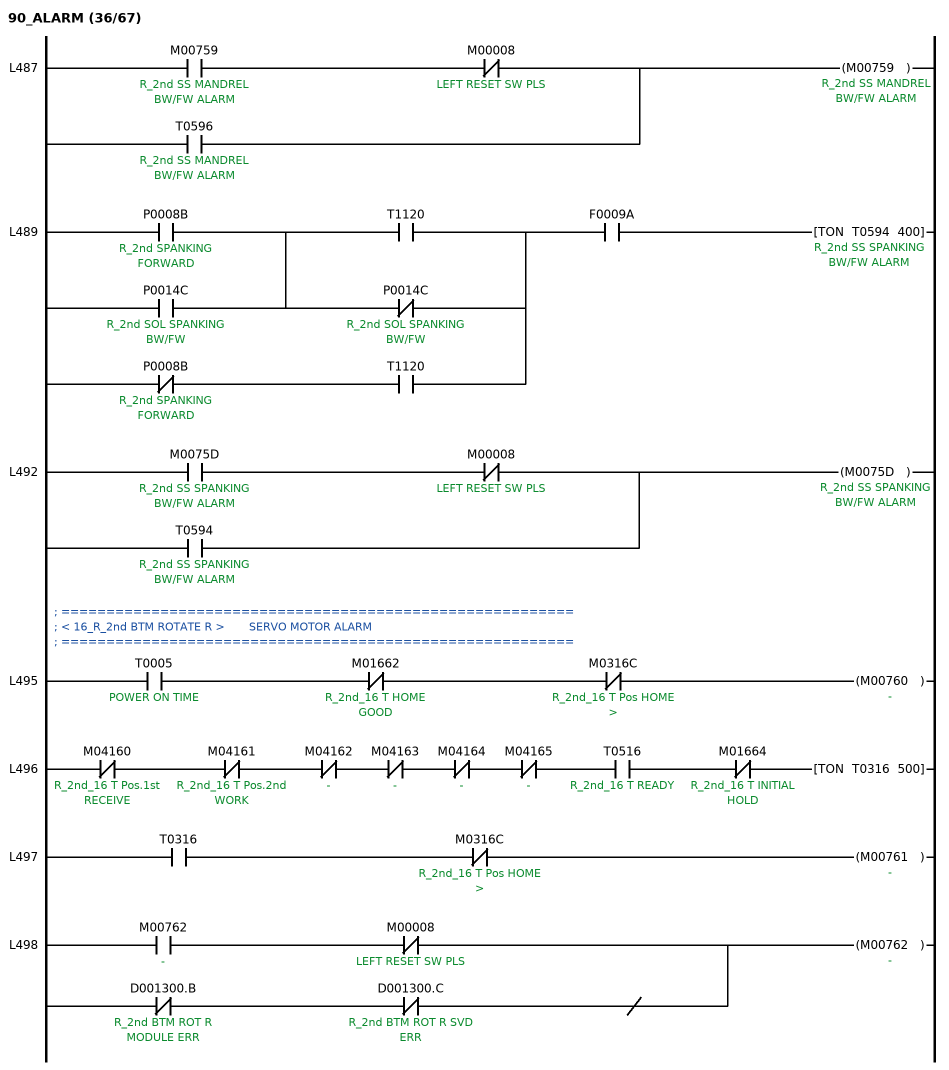
[picture p432: 90_ALARM rungs L487-L498]
; L487
LOAD      M00759	// R_2nd SS MANDREL BW/FW ALARM
AND NOT   M00008	// LEFT RESET SW PLS
OR        T0596	// R_2nd SS MANDREL BW/FW ALARM
OUT       M00759	// R_2nd SS MANDREL BW/FW ALARM
; L489
LOAD      P0008B	// R_2nd SPANKING FORWARD
OR        P0014C	// R_2nd SOL SPANKING BW/FW
LOAD      T1120
OR NOT    P0014C	// R_2nd SOL SPANKING BW/FW
AND LOAD
LOAD NOT  P0008B	// R_2nd SPANKING FORWARD
AND       T1120
OR LOAD
AND       F0009A
TON       T0594 400	// R_2nd SS SPANKING BW/FW ALARM
; L492
LOAD      M0075D	// R_2nd SS SPANKING BW/FW ALARM
AND NOT   M00008	// LEFT RESET SW PLS
OR        T0594	// R_2nd SS SPANKING BW/FW ALARM
OUT       M0075D	// R_2nd SS SPANKING BW/FW ALARM
// =========================================================
// 
//        < 16_R_2nd BTM ROTATE R >       SERVO MOTOR ALARM
// 
// =========================================================
; L495
LOAD      T0005	// POWER ON TIME
AND NOT   M01662	// R_2nd_16 T HOME GOOD
AND NOT   M0316C	// R_2nd_16 T Pos HOME >
OUT       M00760	// -
; L496
LOAD NOT  M04160	// R_2nd_16 T Pos.1st RECEIVE
AND NOT   M04161	// R_2nd_16 T Pos.2nd WORK
AND NOT   M04162	// -
AND NOT   M04163	// -
AND NOT   M04164	// -
AND NOT   M04165	// -
AND       T0516	// R_2nd_16 T READY
AND NOT   M01664	// R_2nd_16 T INITIAL HOLD
TON       T0316 500
; L497
LOAD      T0316
AND NOT   M0316C	// R_2nd_16 T Pos HOME >
OUT       M00761	// -
; L498
LOAD      M00762	// -
AND NOT   M00008	// LEFT RESET SW PLS
LOAD NOT  D001300.B	// R_2nd BTM ROT R MODULE ERR
AND NOT   D001300.C	// R_2nd BTM ROT R SVD ERR
NOT
OR LOAD
OUT       M00762	// -

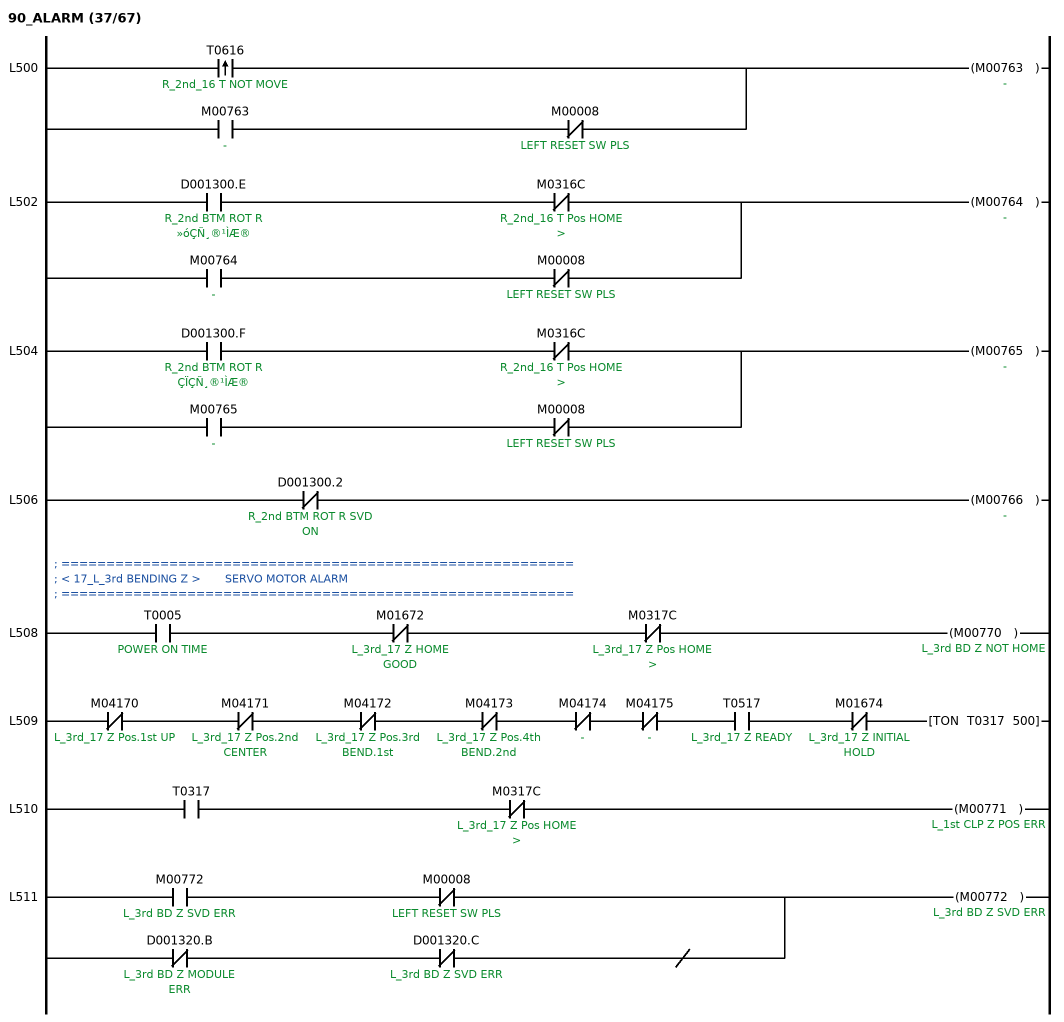
; L500
LOADP     T0616	// R_2nd_16 T NOT MOVE
LOAD      M00763	// -
AND NOT   M00008	// LEFT RESET SW PLS
OR LOAD
OUT       M00763	// -
; L502
LOAD      D001300.E	// R_2nd BTM ROT R »óÇÑ¸®¹ÌÆ®
AND NOT   M0316C	// R_2nd_16 T Pos HOME >
LOAD      M00764	// -
AND NOT   M00008	// LEFT RESET SW PLS
OR LOAD
OUT       M00764	// -
; L504
LOAD      D001300.F	// R_2nd BTM ROT R ÇÏÇÑ¸®¹ÌÆ®
AND NOT   M0316C	// R_2nd_16 T Pos HOME >
LOAD      M00765	// -
AND NOT   M00008	// LEFT RESET SW PLS
OR LOAD
OUT       M00765	// -
; L506
LOAD NOT  D001300.2	// R_2nd BTM ROT R SVD ON
OUT       M00766	// -
// =========================================================
// 
//        < 17_L_3rd BENDING Z >       SERVO MOTOR ALARM
// 
// =========================================================
; L508
LOAD      T0005	// POWER ON TIME
AND NOT   M01672	// L_3rd_17 Z HOME GOOD
AND NOT   M0317C	// L_3rd_17 Z Pos HOME >
OUT       M00770	// L_3rd BD Z NOT HOME
; L509
LOAD NOT  M04170	// L_3rd_17 Z Pos.1st UP
AND NOT   M04171	// L_3rd_17 Z Pos.2nd CENTER
AND NOT   M04172	// L_3rd_17 Z Pos.3rd BEND.1st
AND NOT   M04173	// L_3rd_17 Z Pos.4th BEND.2nd
AND NOT   M04174	// -
AND NOT   M04175	// -
AND       T0517	// L_3rd_17 Z READY
AND NOT   M01674	// L_3rd_17 Z INITIAL HOLD
TON       T0317 500
; L510
LOAD      T0317
AND NOT   M0317C	// L_3rd_17 Z Pos HOME >
OUT       M00771	// L_1st CLP Z POS ERR
; L511
LOAD      M00772	// L_3rd BD Z SVD ERR
AND NOT   M00008	// LEFT RESET SW PLS
LOAD NOT  D001320.B	// L_3rd BD Z MODULE ERR
AND NOT   D001320.C	// L_3rd BD Z SVD ERR
NOT
OR LOAD
OUT       M00772	// L_3rd BD Z SVD ERR

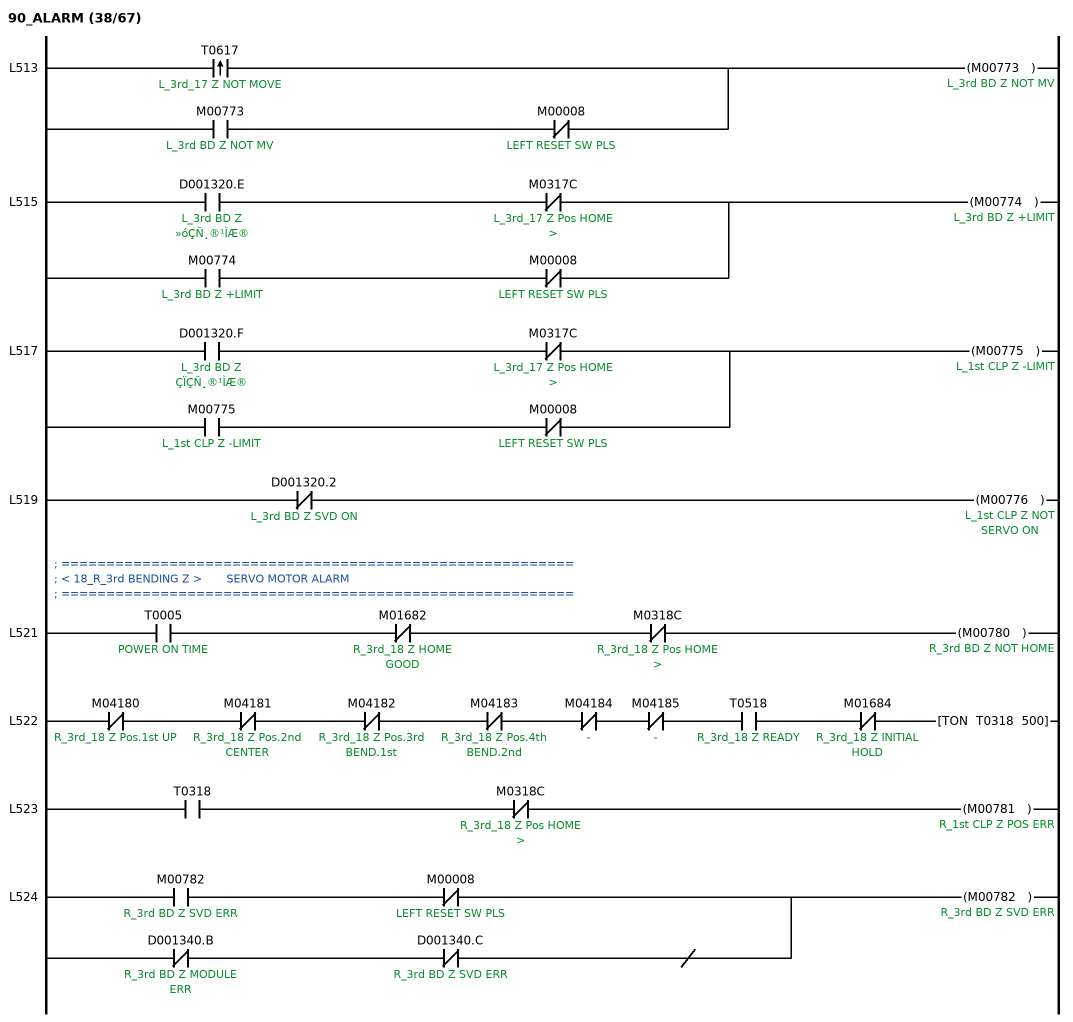
; L513
LOADP     T0617	// L_3rd_17 Z NOT MOVE
LOAD      M00773	// L_3rd BD Z NOT MV
AND NOT   M00008	// LEFT RESET SW PLS
OR LOAD
OUT       M00773	// L_3rd BD Z NOT MV
; L515
LOAD      D001320.E	// L_3rd BD Z »óÇÑ¸®¹ÌÆ®
AND NOT   M0317C	// L_3rd_17 Z Pos HOME >
LOAD      M00774	// L_3rd BD Z +LIMIT
AND NOT   M00008	// LEFT RESET SW PLS
OR LOAD
OUT       M00774	// L_3rd BD Z +LIMIT
; L517
LOAD      D001320.F	// L_3rd BD Z ÇÏÇÑ¸®¹ÌÆ®
AND NOT   M0317C	// L_3rd_17 Z Pos HOME >
LOAD      M00775	// L_1st CLP Z -LIMIT
AND NOT   M00008	// LEFT RESET SW PLS
OR LOAD
OUT       M00775	// L_1st CLP Z -LIMIT
; L519
LOAD NOT  D001320.2	// L_3rd BD Z SVD ON
OUT       M00776	// L_1st CLP Z NOT SERVO ON
// =========================================================
// 
//        < 18_R_3rd BENDING Z >       SERVO MOTOR ALARM
// 
// =========================================================
; L521
LOAD      T0005	// POWER ON TIME
AND NOT   M01682	// R_3rd_18 Z HOME GOOD
AND NOT   M0318C	// R_3rd_18 Z Pos HOME >
OUT       M00780	// R_3rd BD Z NOT HOME
; L522
LOAD NOT  M04180	// R_3rd_18 Z Pos.1st UP
AND NOT   M04181	// R_3rd_18 Z Pos.2nd CENTER
AND NOT   M04182	// R_3rd_18 Z Pos.3rd BEND.1st
AND NOT   M04183	// R_3rd_18 Z Pos.4th BEND.2nd
AND NOT   M04184	// -
AND NOT   M04185	// -
AND       T0518	// R_3rd_18 Z READY
AND NOT   M01684	// R_3rd_18 Z INITIAL HOLD
TON       T0318 500
; L523
LOAD      T0318
AND NOT   M0318C	// R_3rd_18 Z Pos HOME >
OUT       M00781	// R_1st CLP Z POS ERR
; L524
LOAD      M00782	// R_3rd BD Z SVD ERR
AND NOT   M00008	// LEFT RESET SW PLS
LOAD NOT  D001340.B	// R_3rd BD Z MODULE ERR
AND NOT   D001340.C	// R_3rd BD Z SVD ERR
NOT
OR LOAD
OUT       M00782	// R_3rd BD Z SVD ERR

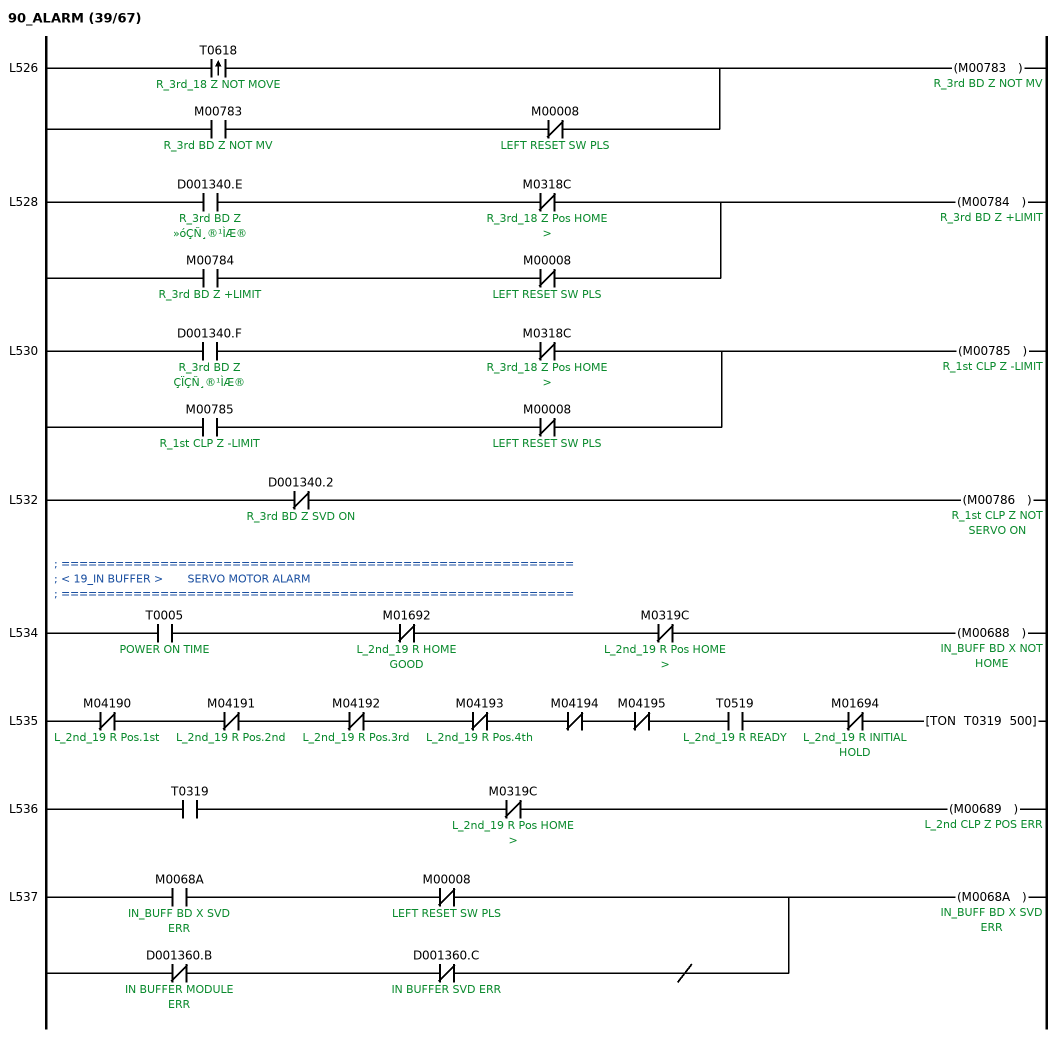
; L526
LOADP     T0618	// R_3rd_18 Z NOT MOVE
LOAD      M00783	// R_3rd BD Z NOT MV
AND NOT   M00008	// LEFT RESET SW PLS
OR LOAD
OUT       M00783	// R_3rd BD Z NOT MV
; L528
LOAD      D001340.E	// R_3rd BD Z »óÇÑ¸®¹ÌÆ®
AND NOT   M0318C	// R_3rd_18 Z Pos HOME >
LOAD      M00784	// R_3rd BD Z +LIMIT
AND NOT   M00008	// LEFT RESET SW PLS
OR LOAD
OUT       M00784	// R_3rd BD Z +LIMIT
; L530
LOAD      D001340.F	// R_3rd BD Z ÇÏÇÑ¸®¹ÌÆ®
AND NOT   M0318C	// R_3rd_18 Z Pos HOME >
LOAD      M00785	// R_1st CLP Z -LIMIT
AND NOT   M00008	// LEFT RESET SW PLS
OR LOAD
OUT       M00785	// R_1st CLP Z -LIMIT
; L532
LOAD NOT  D001340.2	// R_3rd BD Z SVD ON
OUT       M00786	// R_1st CLP Z NOT SERVO ON
// =========================================================
// 
//        < 19_IN BUFFER >       SERVO MOTOR ALARM
// 
// =========================================================
; L534
LOAD      T0005	// POWER ON TIME
AND NOT   M01692	// L_2nd_19 R HOME GOOD
AND NOT   M0319C	// L_2nd_19 R Pos HOME >
OUT       M00688	// IN_BUFF BD X NOT HOME
; L535
LOAD NOT  M04190	// L_2nd_19 R Pos.1st 
AND NOT   M04191	// L_2nd_19 R Pos.2nd
AND NOT   M04192	// L_2nd_19 R Pos.3rd
AND NOT   M04193	// L_2nd_19 R Pos.4th 
AND NOT   M04194
AND NOT   M04195
AND       T0519	// L_2nd_19 R READY
AND NOT   M01694	// L_2nd_19 R INITIAL HOLD
TON       T0319 500
; L536
LOAD      T0319
AND NOT   M0319C	// L_2nd_19 R Pos HOME >
OUT       M00689	// L_2nd CLP Z POS ERR
; L537
LOAD      M0068A	// IN_BUFF BD X SVD ERR
AND NOT   M00008	// LEFT RESET SW PLS
LOAD NOT  D001360.B	// IN BUFFER MODULE ERR
AND NOT   D001360.C	// IN BUFFER SVD ERR
NOT
OR LOAD
OUT       M0068A	// IN_BUFF BD X SVD ERR

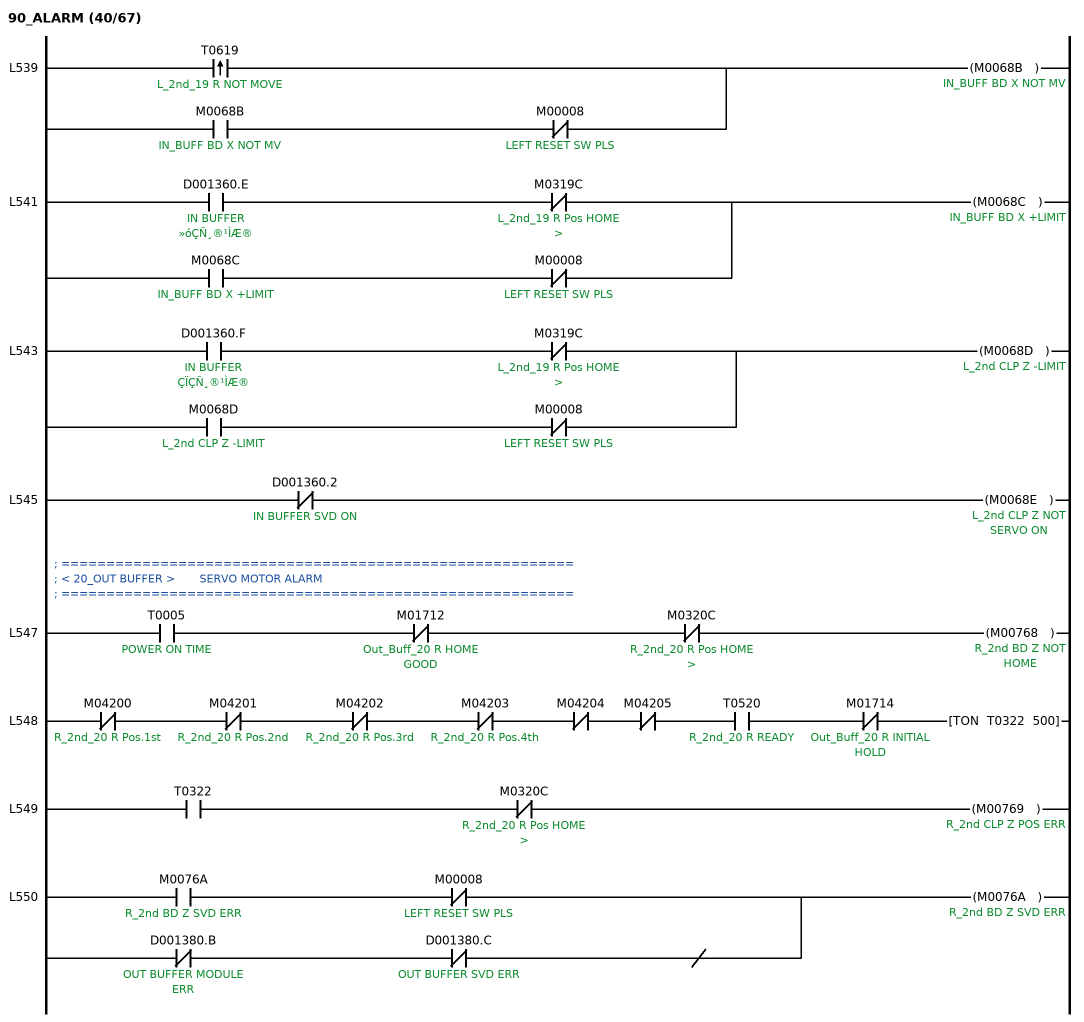
; L539
LOADP     T0619	// L_2nd_19 R NOT MOVE
LOAD      M0068B	// IN_BUFF BD X NOT MV
AND NOT   M00008	// LEFT RESET SW PLS
OR LOAD
OUT       M0068B	// IN_BUFF BD X NOT MV
; L541
LOAD      D001360.E	// IN BUFFER »óÇÑ¸®¹ÌÆ®
AND NOT   M0319C	// L_2nd_19 R Pos HOME >
LOAD      M0068C	// IN_BUFF BD X +LIMIT
AND NOT   M00008	// LEFT RESET SW PLS
OR LOAD
OUT       M0068C	// IN_BUFF BD X +LIMIT
; L543
LOAD      D001360.F	// IN BUFFER ÇÏÇÑ¸®¹ÌÆ®
AND NOT   M0319C	// L_2nd_19 R Pos HOME >
LOAD      M0068D	// L_2nd CLP Z -LIMIT
AND NOT   M00008	// LEFT RESET SW PLS
OR LOAD
OUT       M0068D	// L_2nd CLP Z -LIMIT
; L545
LOAD NOT  D001360.2	// IN BUFFER SVD ON
OUT       M0068E	// L_2nd CLP Z NOT SERVO ON
// =========================================================
// 
//        < 20_OUT BUFFER >       SERVO MOTOR ALARM
// 
// =========================================================
; L547
LOAD      T0005	// POWER ON TIME
AND NOT   M01712	// Out_Buff_20 R HOME GOOD
AND NOT   M0320C	// R_2nd_20 R Pos HOME >
OUT       M00768	// R_2nd BD Z NOT HOME
; L548
LOAD NOT  M04200	// R_2nd_20 R Pos.1st
AND NOT   M04201	// R_2nd_20 R Pos.2nd
AND NOT   M04202	// R_2nd_20 R Pos.3rd
AND NOT   M04203	// R_2nd_20 R Pos.4th 
AND NOT   M04204
AND NOT   M04205
AND       T0520	// R_2nd_20 R READY
AND NOT   M01714	// Out_Buff_20 R INITIAL HOLD
TON       T0322 500
; L549
LOAD      T0322
AND NOT   M0320C	// R_2nd_20 R Pos HOME >
OUT       M00769	// R_2nd CLP Z POS ERR
; L550
LOAD      M0076A	// R_2nd BD Z SVD ERR
AND NOT   M00008	// LEFT RESET SW PLS
LOAD NOT  D001380.B	// OUT BUFFER MODULE ERR
AND NOT   D001380.C	// OUT BUFFER SVD ERR
NOT
OR LOAD
OUT       M0076A	// R_2nd BD Z SVD ERR

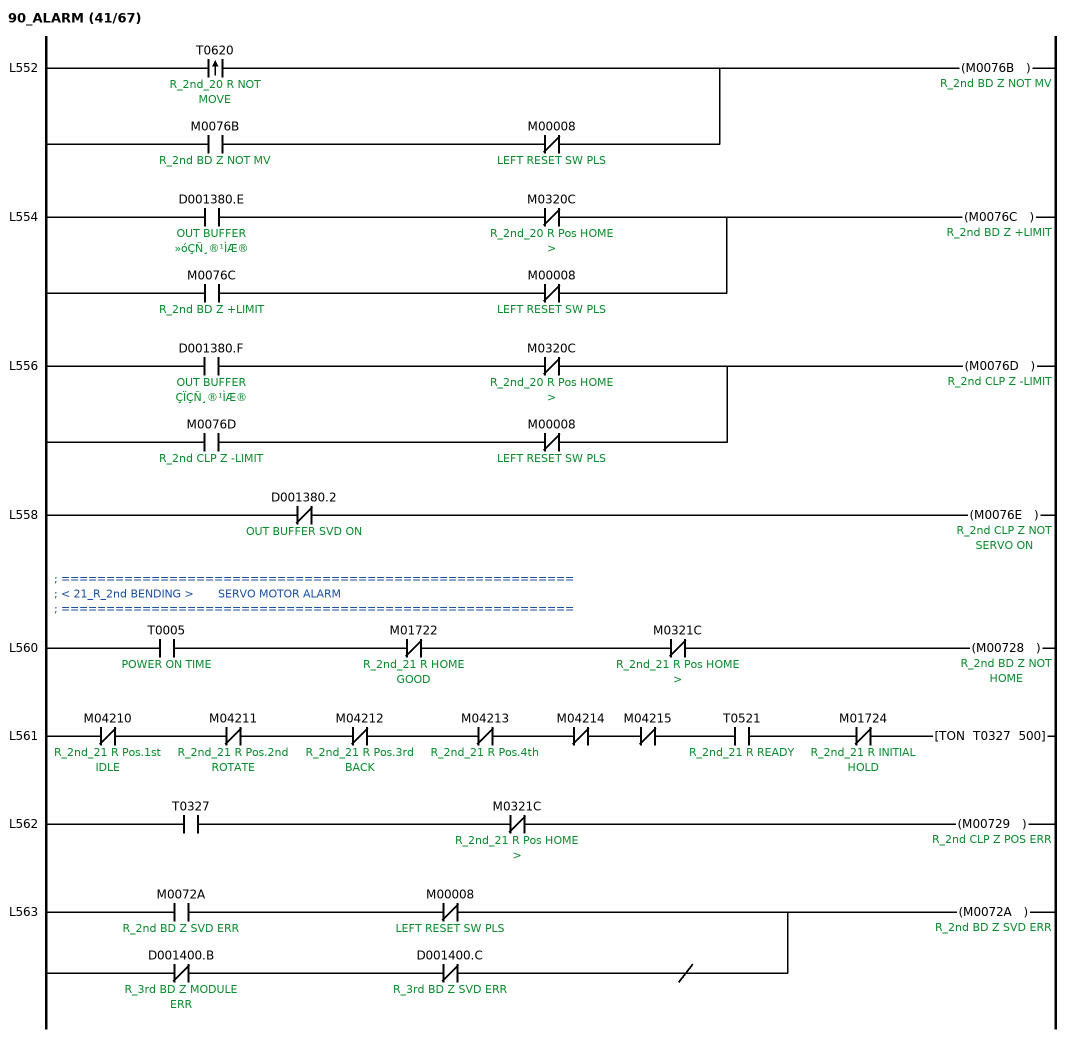
; L552
LOADP     T0620	// R_2nd_20 R NOT MOVE
LOAD      M0076B	// R_2nd BD Z NOT MV
AND NOT   M00008	// LEFT RESET SW PLS
OR LOAD
OUT       M0076B	// R_2nd BD Z NOT MV
; L554
LOAD      D001380.E	// OUT BUFFER »óÇÑ¸®¹ÌÆ®
AND NOT   M0320C	// R_2nd_20 R Pos HOME >
LOAD      M0076C	// R_2nd BD Z +LIMIT
AND NOT   M00008	// LEFT RESET SW PLS
OR LOAD
OUT       M0076C	// R_2nd BD Z +LIMIT
; L556
LOAD      D001380.F	// OUT BUFFER ÇÏÇÑ¸®¹ÌÆ®
AND NOT   M0320C	// R_2nd_20 R Pos HOME >
LOAD      M0076D	// R_2nd CLP Z -LIMIT
AND NOT   M00008	// LEFT RESET SW PLS
OR LOAD
OUT       M0076D	// R_2nd CLP Z -LIMIT
; L558
LOAD NOT  D001380.2	// OUT BUFFER SVD ON
OUT       M0076E	// R_2nd CLP Z NOT SERVO ON
// =========================================================
// 
//        < 21_R_2nd BENDING >       SERVO MOTOR ALARM
// 
// =========================================================
; L560
LOAD      T0005	// POWER ON TIME
AND NOT   M01722	// R_2nd_21 R HOME GOOD
AND NOT   M0321C	// R_2nd_21 R Pos HOME >
OUT       M00728	// R_2nd BD Z NOT HOME
; L561
LOAD NOT  M04210	// R_2nd_21 R Pos.1st IDLE
AND NOT   M04211	// R_2nd_21 R Pos.2nd ROTATE
AND NOT   M04212	// R_2nd_21 R Pos.3rd BACK
AND NOT   M04213	// R_2nd_21 R Pos.4th 
AND NOT   M04214
AND NOT   M04215
AND       T0521	// R_2nd_21 R READY
AND NOT   M01724	// R_2nd_21 R INITIAL HOLD
TON       T0327 500
; L562
LOAD      T0327
AND NOT   M0321C	// R_2nd_21 R Pos HOME >
OUT       M00729	// R_2nd CLP Z POS ERR
; L563
LOAD      M0072A	// R_2nd BD Z SVD ERR
AND NOT   M00008	// LEFT RESET SW PLS
LOAD NOT  D001400.B	// R_3rd BD Z MODULE ERR
AND NOT   D001400.C	// R_3rd BD Z SVD ERR
NOT
OR LOAD
OUT       M0072A	// R_2nd BD Z SVD ERR

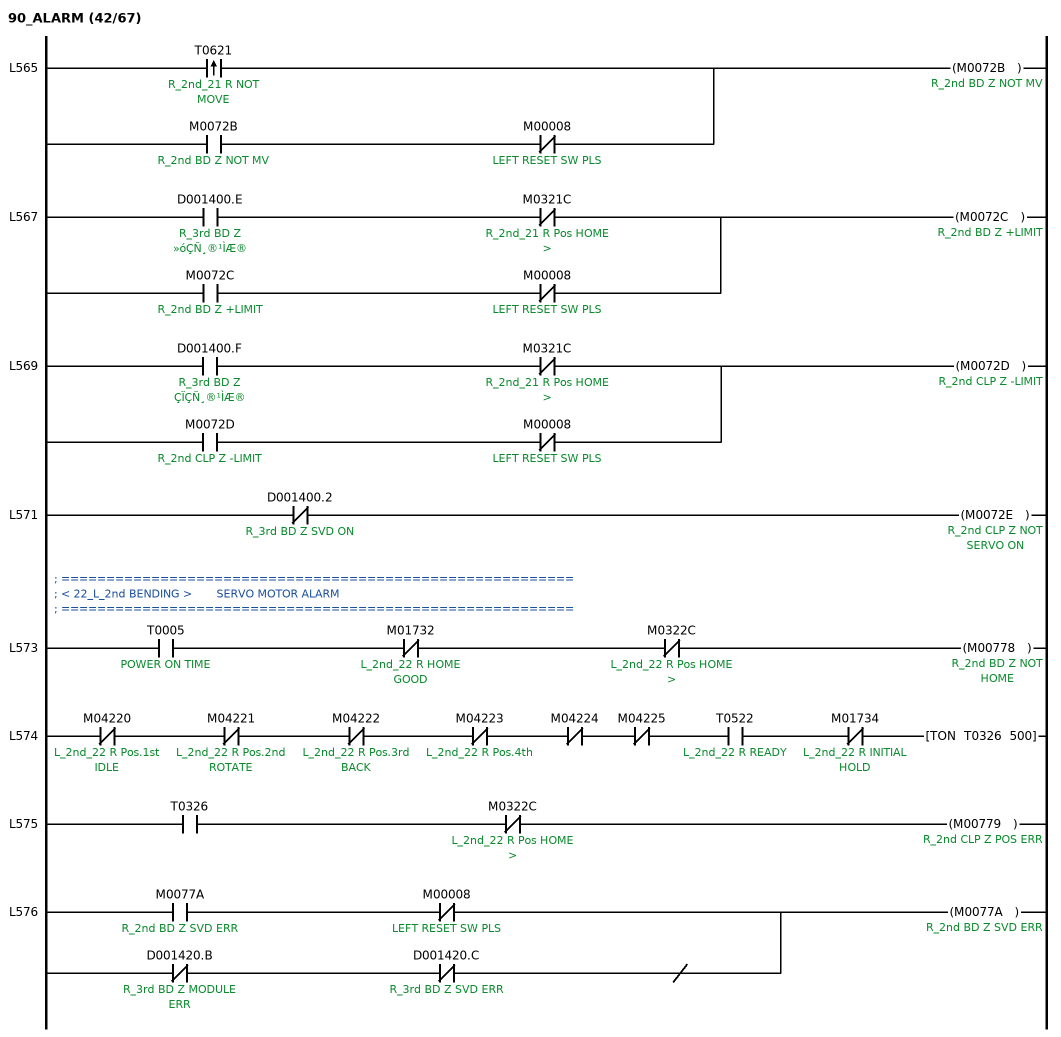
; L565
LOADP     T0621	// R_2nd_21 R NOT MOVE
LOAD      M0072B	// R_2nd BD Z NOT MV
AND NOT   M00008	// LEFT RESET SW PLS
OR LOAD
OUT       M0072B	// R_2nd BD Z NOT MV
; L567
LOAD      D001400.E	// R_3rd BD Z »óÇÑ¸®¹ÌÆ®
AND NOT   M0321C	// R_2nd_21 R Pos HOME >
LOAD      M0072C	// R_2nd BD Z +LIMIT
AND NOT   M00008	// LEFT RESET SW PLS
OR LOAD
OUT       M0072C	// R_2nd BD Z +LIMIT
; L569
LOAD      D001400.F	// R_3rd BD Z ÇÏÇÑ¸®¹ÌÆ®
AND NOT   M0321C	// R_2nd_21 R Pos HOME >
LOAD      M0072D	// R_2nd CLP Z -LIMIT
AND NOT   M00008	// LEFT RESET SW PLS
OR LOAD
OUT       M0072D	// R_2nd CLP Z -LIMIT
; L571
LOAD NOT  D001400.2	// R_3rd BD Z SVD ON
OUT       M0072E	// R_2nd CLP Z NOT SERVO ON
// =========================================================
// 
//        < 22_L_2nd BENDING >       SERVO MOTOR ALARM
// 
// =========================================================
; L573
LOAD      T0005	// POWER ON TIME
AND NOT   M01732	// L_2nd_22 R HOME GOOD
AND NOT   M0322C	// L_2nd_22 R Pos HOME >
OUT       M00778	// R_2nd BD Z NOT HOME
; L574
LOAD NOT  M04220	// L_2nd_22 R Pos.1st IDLE
AND NOT   M04221	// L_2nd_22 R Pos.2nd ROTATE
AND NOT   M04222	// L_2nd_22 R Pos.3rd BACK
AND NOT   M04223	// L_2nd_22 R Pos.4th 
AND NOT   M04224
AND NOT   M04225
AND       T0522	// L_2nd_22 R READY
AND NOT   M01734	// L_2nd_22 R INITIAL HOLD
TON       T0326 500
; L575
LOAD      T0326
AND NOT   M0322C	// L_2nd_22 R Pos HOME >
OUT       M00779	// R_2nd CLP Z POS ERR
; L576
LOAD      M0077A	// R_2nd BD Z SVD ERR
AND NOT   M00008	// LEFT RESET SW PLS
LOAD NOT  D001420.B	// R_3rd BD Z MODULE ERR
AND NOT   D001420.C	// R_3rd BD Z SVD ERR
NOT
OR LOAD
OUT       M0077A	// R_2nd BD Z SVD ERR

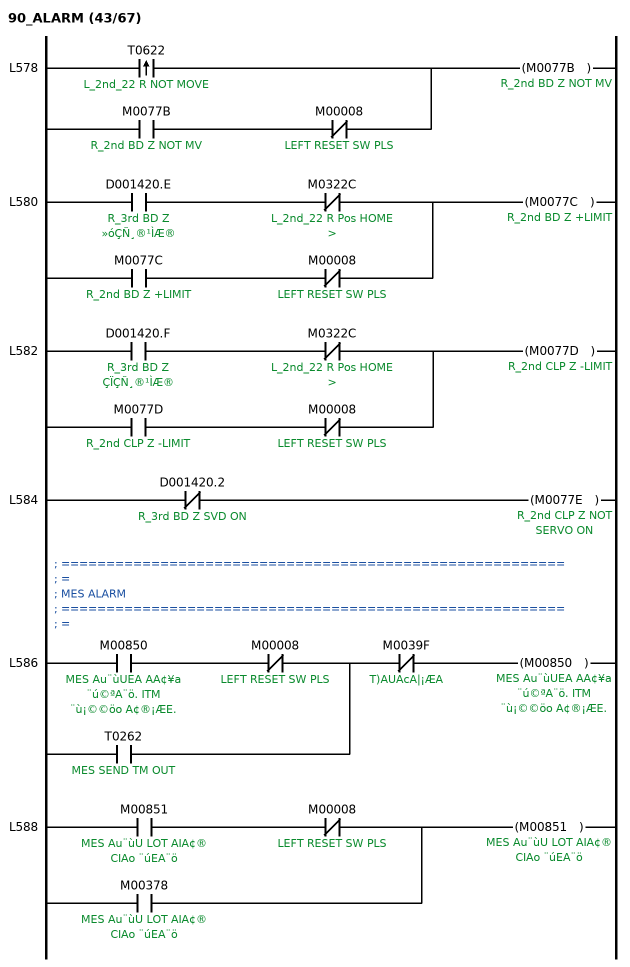
; L578
LOADP     T0622	// L_2nd_22 R NOT MOVE
LOAD      M0077B	// R_2nd BD Z NOT MV
AND NOT   M00008	// LEFT RESET SW PLS
OR LOAD
OUT       M0077B	// R_2nd BD Z NOT MV
; L580
LOAD      D001420.E	// R_3rd BD Z »óÇÑ¸®¹ÌÆ®
AND NOT   M0322C	// L_2nd_22 R Pos HOME >
LOAD      M0077C	// R_2nd BD Z +LIMIT
AND NOT   M00008	// LEFT RESET SW PLS
OR LOAD
OUT       M0077C	// R_2nd BD Z +LIMIT
; L582
LOAD      D001420.F	// R_3rd BD Z ÇÏÇÑ¸®¹ÌÆ®
AND NOT   M0322C	// L_2nd_22 R Pos HOME >
LOAD      M0077D	// R_2nd CLP Z -LIMIT
AND NOT   M00008	// LEFT RESET SW PLS
OR LOAD
OUT       M0077D	// R_2nd CLP Z -LIMIT
; L584
LOAD NOT  D001420.2	// R_3rd BD Z SVD ON
OUT       M0077E	// R_2nd CLP Z NOT SERVO ON
// =========================================================
// 
//        MES ALARM
// 
// =========================================================
; L586
LOAD      M00850	// MES Au¨ùUEA AA¢¥a ¨ú©ªA¨ö. ITM ¨ù¡©©öo A¢®¡ÆE.
AND NOT   M00008	// LEFT RESET SW PLS
OR        T0262	// MES SEND TM OUT
AND NOT   M0039F	// T)AUAcA|¡ÆA
OUT       M00850	// MES Au¨ùUEA AA¢¥a ¨ú©ªA¨ö. ITM ¨ù¡©©öo A¢®¡ÆE.
; L588
LOAD      M00851	// MES Au¨ùU LOT AIA¢® CIAo ¨úEA¨ö
AND NOT   M00008	// LEFT RESET SW PLS
OR        M00378	// MES Au¨ùU LOT AIA¢® CIAo ¨úEA¨ö
OUT       M00851	// MES Au¨ùU LOT AIA¢® CIAo ¨úEA¨ö

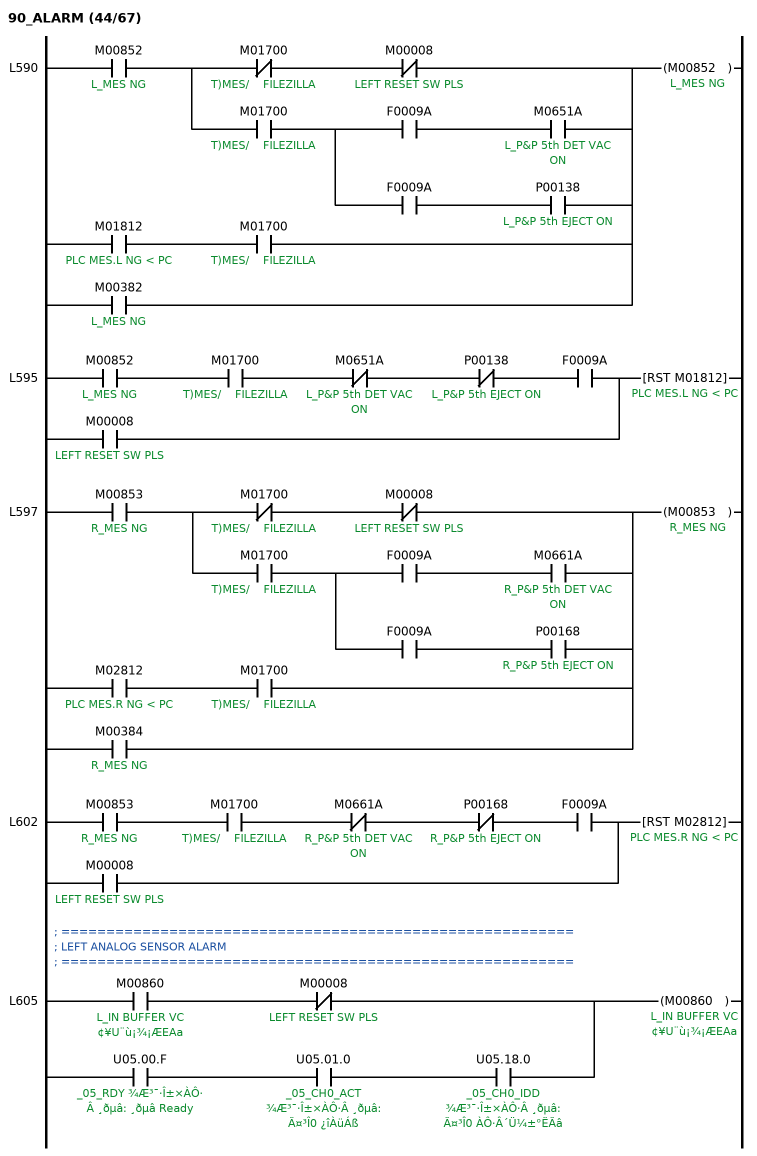
; L590
LOAD      M00852	// L_MES NG
LOAD NOT  M01700	// T)MES/    FILEZILLA
AND NOT   M00008	// LEFT RESET SW PLS
LOAD      M01700	// T)MES/    FILEZILLA
LOAD      F0009A
AND       M0651A	// L_P&P 5th DET VAC ON
LOAD      F0009A
AND       P00138	// L_P&P 5th EJECT ON
OR LOAD
AND LOAD
OR LOAD
AND LOAD
LOAD      M01812	// PLC MES.L NG < PC
AND       M01700	// T)MES/    FILEZILLA
OR LOAD
OR        M00382	// L_MES NG
OUT       M00852	// L_MES NG
; L595
LOAD      M00852	// L_MES NG
AND       M01700	// T)MES/    FILEZILLA
AND NOT   M0651A	// L_P&P 5th DET VAC ON
AND NOT   P00138	// L_P&P 5th EJECT ON
AND       F0009A
OR        M00008	// LEFT RESET SW PLS
RST       M01812	// PLC MES.L NG < PC
; L597
LOAD      M00853	// R_MES NG
LOAD NOT  M01700	// T)MES/    FILEZILLA
AND NOT   M00008	// LEFT RESET SW PLS
LOAD      M01700	// T)MES/    FILEZILLA
LOAD      F0009A
AND       M0661A	// R_P&P 5th DET VAC ON
LOAD      F0009A
AND       P00168	// R_P&P 5th EJECT ON
OR LOAD
AND LOAD
OR LOAD
AND LOAD
LOAD      M02812	// PLC MES.R NG < PC
AND       M01700	// T)MES/    FILEZILLA
OR LOAD
OR        M00384	// R_MES NG
OUT       M00853	// R_MES NG
; L602
LOAD      M00853	// R_MES NG
AND       M01700	// T)MES/    FILEZILLA
AND NOT   M0661A	// R_P&P 5th DET VAC ON
AND NOT   P00168	// R_P&P 5th EJECT ON
AND       F0009A
OR        M00008	// LEFT RESET SW PLS
RST       M02812	// PLC MES.R NG < PC
// =========================================================
// 
//        LEFT ANALOG SENSOR ALARM
// 
// =========================================================
; L605
LOAD      M00860	// L_IN BUFFER VC ¢¥U¨ù¡¾¡ÆEAa
AND NOT   M00008	// LEFT RESET SW PLS
LOAD      U05.00.F	// _05_RDY ¾Æ³¯·Î±×ÀÔ·Â ¸ðµâ: ¸ðµâ Ready
AND       U05.01.0	// _05_CH0_ACT ¾Æ³¯·Î±×ÀÔ·Â ¸ðµâ: Ã¤³Î0 ¿îÀüÁß
AND       U05.18.0	// _05_CH0_IDD ¾Æ³¯·Î±×ÀÔ·Â ¸ðµâ: Ã¤³Î0 ÀÔ·Â´Ü¼±°ËÃâ
OR LOAD
OUT       M00860	// L_IN BUFFER VC ¢¥U¨ù¡¾¡ÆEAa

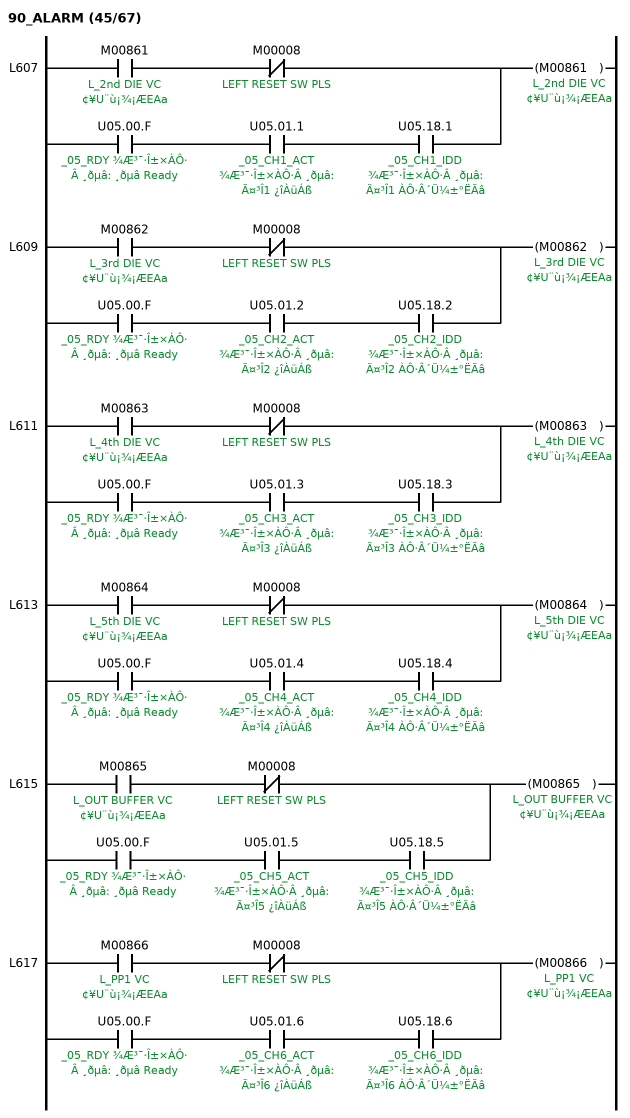
; L607
LOAD      M00861	// L_2nd DIE VC ¢¥U¨ù¡¾¡ÆEAa
AND NOT   M00008	// LEFT RESET SW PLS
LOAD      U05.00.F	// _05_RDY ¾Æ³¯·Î±×ÀÔ·Â ¸ðµâ: ¸ðµâ Ready
AND       U05.01.1	// _05_CH1_ACT ¾Æ³¯·Î±×ÀÔ·Â ¸ðµâ: Ã¤³Î1 ¿îÀüÁß
AND       U05.18.1	// _05_CH1_IDD ¾Æ³¯·Î±×ÀÔ·Â ¸ðµâ: Ã¤³Î1 ÀÔ·Â´Ü¼±°ËÃâ
OR LOAD
OUT       M00861	// L_2nd DIE VC ¢¥U¨ù¡¾¡ÆEAa
; L609
LOAD      M00862	// L_3rd DIE VC ¢¥U¨ù¡¾¡ÆEAa
AND NOT   M00008	// LEFT RESET SW PLS
LOAD      U05.00.F	// _05_RDY ¾Æ³¯·Î±×ÀÔ·Â ¸ðµâ: ¸ðµâ Ready
AND       U05.01.2	// _05_CH2_ACT ¾Æ³¯·Î±×ÀÔ·Â ¸ðµâ: Ã¤³Î2 ¿îÀüÁß
AND       U05.18.2	// _05_CH2_IDD ¾Æ³¯·Î±×ÀÔ·Â ¸ðµâ: Ã¤³Î2 ÀÔ·Â´Ü¼±°ËÃâ
OR LOAD
OUT       M00862	// L_3rd DIE VC ¢¥U¨ù¡¾¡ÆEAa
; L611
LOAD      M00863	// L_4th DIE VC ¢¥U¨ù¡¾¡ÆEAa
AND NOT   M00008	// LEFT RESET SW PLS
LOAD      U05.00.F	// _05_RDY ¾Æ³¯·Î±×ÀÔ·Â ¸ðµâ: ¸ðµâ Ready
AND       U05.01.3	// _05_CH3_ACT ¾Æ³¯·Î±×ÀÔ·Â ¸ðµâ: Ã¤³Î3 ¿îÀüÁß
AND       U05.18.3	// _05_CH3_IDD ¾Æ³¯·Î±×ÀÔ·Â ¸ðµâ: Ã¤³Î3 ÀÔ·Â´Ü¼±°ËÃâ
OR LOAD
OUT       M00863	// L_4th DIE VC ¢¥U¨ù¡¾¡ÆEAa
; L613
LOAD      M00864	// L_5th DIE VC ¢¥U¨ù¡¾¡ÆEAa
AND NOT   M00008	// LEFT RESET SW PLS
LOAD      U05.00.F	// _05_RDY ¾Æ³¯·Î±×ÀÔ·Â ¸ðµâ: ¸ðµâ Ready
AND       U05.01.4	// _05_CH4_ACT ¾Æ³¯·Î±×ÀÔ·Â ¸ðµâ: Ã¤³Î4 ¿îÀüÁß
AND       U05.18.4	// _05_CH4_IDD ¾Æ³¯·Î±×ÀÔ·Â ¸ðµâ: Ã¤³Î4 ÀÔ·Â´Ü¼±°ËÃâ
OR LOAD
OUT       M00864	// L_5th DIE VC ¢¥U¨ù¡¾¡ÆEAa
; L615
LOAD      M00865	// L_OUT BUFFER VC ¢¥U¨ù¡¾¡ÆEAa
AND NOT   M00008	// LEFT RESET SW PLS
LOAD      U05.00.F	// _05_RDY ¾Æ³¯·Î±×ÀÔ·Â ¸ðµâ: ¸ðµâ Ready
AND       U05.01.5	// _05_CH5_ACT ¾Æ³¯·Î±×ÀÔ·Â ¸ðµâ: Ã¤³Î5 ¿îÀüÁß
AND       U05.18.5	// _05_CH5_IDD ¾Æ³¯·Î±×ÀÔ·Â ¸ðµâ: Ã¤³Î5 ÀÔ·Â´Ü¼±°ËÃâ
OR LOAD
OUT       M00865	// L_OUT BUFFER VC ¢¥U¨ù¡¾¡ÆEAa
; L617
LOAD      M00866	// L_PP1 VC ¢¥U¨ù¡¾¡ÆEAa
AND NOT   M00008	// LEFT RESET SW PLS
LOAD      U05.00.F	// _05_RDY ¾Æ³¯·Î±×ÀÔ·Â ¸ðµâ: ¸ðµâ Ready
AND       U05.01.6	// _05_CH6_ACT ¾Æ³¯·Î±×ÀÔ·Â ¸ðµâ: Ã¤³Î6 ¿îÀüÁß
AND       U05.18.6	// _05_CH6_IDD ¾Æ³¯·Î±×ÀÔ·Â ¸ðµâ: Ã¤³Î6 ÀÔ·Â´Ü¼±°ËÃâ
OR LOAD
OUT       M00866	// L_PP1 VC ¢¥U¨ù¡¾¡ÆEAa

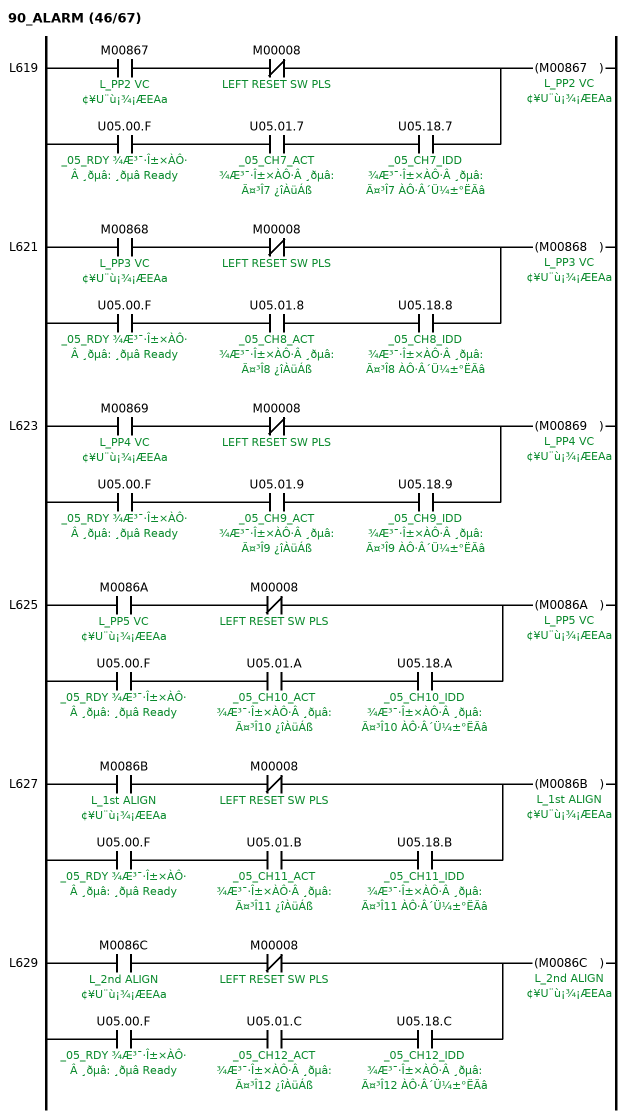
; L619
LOAD      M00867	// L_PP2 VC ¢¥U¨ù¡¾¡ÆEAa
AND NOT   M00008	// LEFT RESET SW PLS
LOAD      U05.00.F	// _05_RDY ¾Æ³¯·Î±×ÀÔ·Â ¸ðµâ: ¸ðµâ Ready
AND       U05.01.7	// _05_CH7_ACT ¾Æ³¯·Î±×ÀÔ·Â ¸ðµâ: Ã¤³Î7 ¿îÀüÁß
AND       U05.18.7	// _05_CH7_IDD ¾Æ³¯·Î±×ÀÔ·Â ¸ðµâ: Ã¤³Î7 ÀÔ·Â´Ü¼±°ËÃâ
OR LOAD
OUT       M00867	// L_PP2 VC ¢¥U¨ù¡¾¡ÆEAa
; L621
LOAD      M00868	// L_PP3 VC ¢¥U¨ù¡¾¡ÆEAa
AND NOT   M00008	// LEFT RESET SW PLS
LOAD      U05.00.F	// _05_RDY ¾Æ³¯·Î±×ÀÔ·Â ¸ðµâ: ¸ðµâ Ready
AND       U05.01.8	// _05_CH8_ACT ¾Æ³¯·Î±×ÀÔ·Â ¸ðµâ: Ã¤³Î8 ¿îÀüÁß
AND       U05.18.8	// _05_CH8_IDD ¾Æ³¯·Î±×ÀÔ·Â ¸ðµâ: Ã¤³Î8 ÀÔ·Â´Ü¼±°ËÃâ
OR LOAD
OUT       M00868	// L_PP3 VC ¢¥U¨ù¡¾¡ÆEAa
; L623
LOAD      M00869	// L_PP4 VC ¢¥U¨ù¡¾¡ÆEAa
AND NOT   M00008	// LEFT RESET SW PLS
LOAD      U05.00.F	// _05_RDY ¾Æ³¯·Î±×ÀÔ·Â ¸ðµâ: ¸ðµâ Ready
AND       U05.01.9	// _05_CH9_ACT ¾Æ³¯·Î±×ÀÔ·Â ¸ðµâ: Ã¤³Î9 ¿îÀüÁß
AND       U05.18.9	// _05_CH9_IDD ¾Æ³¯·Î±×ÀÔ·Â ¸ðµâ: Ã¤³Î9 ÀÔ·Â´Ü¼±°ËÃâ
OR LOAD
OUT       M00869	// L_PP4 VC ¢¥U¨ù¡¾¡ÆEAa
; L625
LOAD      M0086A	// L_PP5 VC ¢¥U¨ù¡¾¡ÆEAa
AND NOT   M00008	// LEFT RESET SW PLS
LOAD      U05.00.F	// _05_RDY ¾Æ³¯·Î±×ÀÔ·Â ¸ðµâ: ¸ðµâ Ready
AND       U05.01.A	// _05_CH10_ACT ¾Æ³¯·Î±×ÀÔ·Â ¸ðµâ: Ã¤³Î10 ¿îÀüÁß
AND       U05.18.A	// _05_CH10_IDD ¾Æ³¯·Î±×ÀÔ·Â ¸ðµâ: Ã¤³Î10 ÀÔ·Â´Ü¼±°ËÃâ
OR LOAD
OUT       M0086A	// L_PP5 VC ¢¥U¨ù¡¾¡ÆEAa
; L627
LOAD      M0086B	// L_1st ALIGN ¢¥U¨ù¡¾¡ÆEAa
AND NOT   M00008	// LEFT RESET SW PLS
LOAD      U05.00.F	// _05_RDY ¾Æ³¯·Î±×ÀÔ·Â ¸ðµâ: ¸ðµâ Ready
AND       U05.01.B	// _05_CH11_ACT ¾Æ³¯·Î±×ÀÔ·Â ¸ðµâ: Ã¤³Î11 ¿îÀüÁß
AND       U05.18.B	// _05_CH11_IDD ¾Æ³¯·Î±×ÀÔ·Â ¸ðµâ: Ã¤³Î11 ÀÔ·Â´Ü¼±°ËÃâ
OR LOAD
OUT       M0086B	// L_1st ALIGN ¢¥U¨ù¡¾¡ÆEAa
; L629
LOAD      M0086C	// L_2nd ALIGN ¢¥U¨ù¡¾¡ÆEAa
AND NOT   M00008	// LEFT RESET SW PLS
LOAD      U05.00.F	// _05_RDY ¾Æ³¯·Î±×ÀÔ·Â ¸ðµâ: ¸ðµâ Ready
AND       U05.01.C	// _05_CH12_ACT ¾Æ³¯·Î±×ÀÔ·Â ¸ðµâ: Ã¤³Î12 ¿îÀüÁß
AND       U05.18.C	// _05_CH12_IDD ¾Æ³¯·Î±×ÀÔ·Â ¸ðµâ: Ã¤³Î12 ÀÔ·Â´Ü¼±°ËÃâ
OR LOAD
OUT       M0086C	// L_2nd ALIGN ¢¥U¨ù¡¾¡ÆEAa

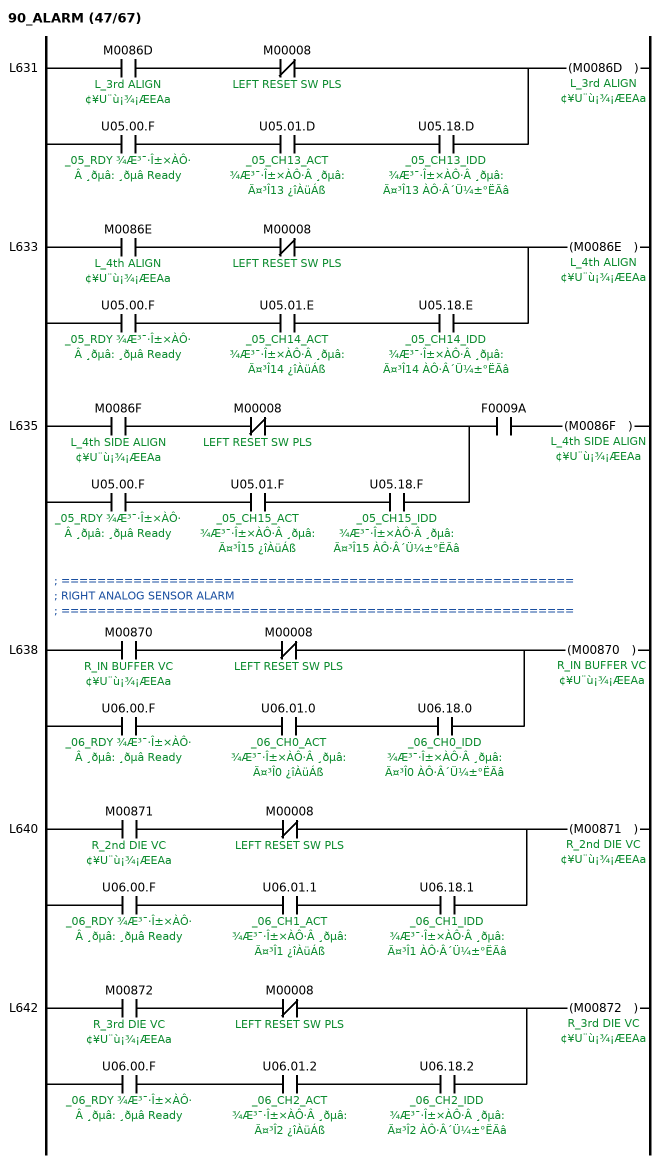
; L631
LOAD      M0086D	// L_3rd ALIGN ¢¥U¨ù¡¾¡ÆEAa
AND NOT   M00008	// LEFT RESET SW PLS
LOAD      U05.00.F	// _05_RDY ¾Æ³¯·Î±×ÀÔ·Â ¸ðµâ: ¸ðµâ Ready
AND       U05.01.D	// _05_CH13_ACT ¾Æ³¯·Î±×ÀÔ·Â ¸ðµâ: Ã¤³Î13 ¿îÀüÁß
AND       U05.18.D	// _05_CH13_IDD ¾Æ³¯·Î±×ÀÔ·Â ¸ðµâ: Ã¤³Î13 ÀÔ·Â´Ü¼±°ËÃâ
OR LOAD
OUT       M0086D	// L_3rd ALIGN ¢¥U¨ù¡¾¡ÆEAa
; L633
LOAD      M0086E	// L_4th ALIGN ¢¥U¨ù¡¾¡ÆEAa
AND NOT   M00008	// LEFT RESET SW PLS
LOAD      U05.00.F	// _05_RDY ¾Æ³¯·Î±×ÀÔ·Â ¸ðµâ: ¸ðµâ Ready
AND       U05.01.E	// _05_CH14_ACT ¾Æ³¯·Î±×ÀÔ·Â ¸ðµâ: Ã¤³Î14 ¿îÀüÁß
AND       U05.18.E	// _05_CH14_IDD ¾Æ³¯·Î±×ÀÔ·Â ¸ðµâ: Ã¤³Î14 ÀÔ·Â´Ü¼±°ËÃâ
OR LOAD
OUT       M0086E	// L_4th ALIGN ¢¥U¨ù¡¾¡ÆEAa
; L635
LOAD      M0086F	// L_4th SIDE ALIGN ¢¥U¨ù¡¾¡ÆEAa
AND NOT   M00008	// LEFT RESET SW PLS
LOAD      U05.00.F	// _05_RDY ¾Æ³¯·Î±×ÀÔ·Â ¸ðµâ: ¸ðµâ Ready
AND       U05.01.F	// _05_CH15_ACT ¾Æ³¯·Î±×ÀÔ·Â ¸ðµâ: Ã¤³Î15 ¿îÀüÁß
AND       U05.18.F	// _05_CH15_IDD ¾Æ³¯·Î±×ÀÔ·Â ¸ðµâ: Ã¤³Î15 ÀÔ·Â´Ü¼±°ËÃâ
OR LOAD
AND       F0009A
OUT       M0086F	// L_4th SIDE ALIGN ¢¥U¨ù¡¾¡ÆEAa
// =========================================================
// 
//        RIGHT ANALOG SENSOR ALARM
// 
// =========================================================
; L638
LOAD      M00870	// R_IN BUFFER VC ¢¥U¨ù¡¾¡ÆEAa
AND NOT   M00008	// LEFT RESET SW PLS
LOAD      U06.00.F	// _06_RDY ¾Æ³¯·Î±×ÀÔ·Â ¸ðµâ: ¸ðµâ Ready
AND       U06.01.0	// _06_CH0_ACT ¾Æ³¯·Î±×ÀÔ·Â ¸ðµâ: Ã¤³Î0 ¿îÀüÁß
AND       U06.18.0	// _06_CH0_IDD ¾Æ³¯·Î±×ÀÔ·Â ¸ðµâ: Ã¤³Î0 ÀÔ·Â´Ü¼±°ËÃâ
OR LOAD
OUT       M00870	// R_IN BUFFER VC ¢¥U¨ù¡¾¡ÆEAa
; L640
LOAD      M00871	// R_2nd DIE VC ¢¥U¨ù¡¾¡ÆEAa
AND NOT   M00008	// LEFT RESET SW PLS
LOAD      U06.00.F	// _06_RDY ¾Æ³¯·Î±×ÀÔ·Â ¸ðµâ: ¸ðµâ Ready
AND       U06.01.1	// _06_CH1_ACT ¾Æ³¯·Î±×ÀÔ·Â ¸ðµâ: Ã¤³Î1 ¿îÀüÁß
AND       U06.18.1	// _06_CH1_IDD ¾Æ³¯·Î±×ÀÔ·Â ¸ðµâ: Ã¤³Î1 ÀÔ·Â´Ü¼±°ËÃâ
OR LOAD
OUT       M00871	// R_2nd DIE VC ¢¥U¨ù¡¾¡ÆEAa
; L642
LOAD      M00872	// R_3rd DIE VC ¢¥U¨ù¡¾¡ÆEAa
AND NOT   M00008	// LEFT RESET SW PLS
LOAD      U06.00.F	// _06_RDY ¾Æ³¯·Î±×ÀÔ·Â ¸ðµâ: ¸ðµâ Ready
AND       U06.01.2	// _06_CH2_ACT ¾Æ³¯·Î±×ÀÔ·Â ¸ðµâ: Ã¤³Î2 ¿îÀüÁß
AND       U06.18.2	// _06_CH2_IDD ¾Æ³¯·Î±×ÀÔ·Â ¸ðµâ: Ã¤³Î2 ÀÔ·Â´Ü¼±°ËÃâ
OR LOAD
OUT       M00872	// R_3rd DIE VC ¢¥U¨ù¡¾¡ÆEAa

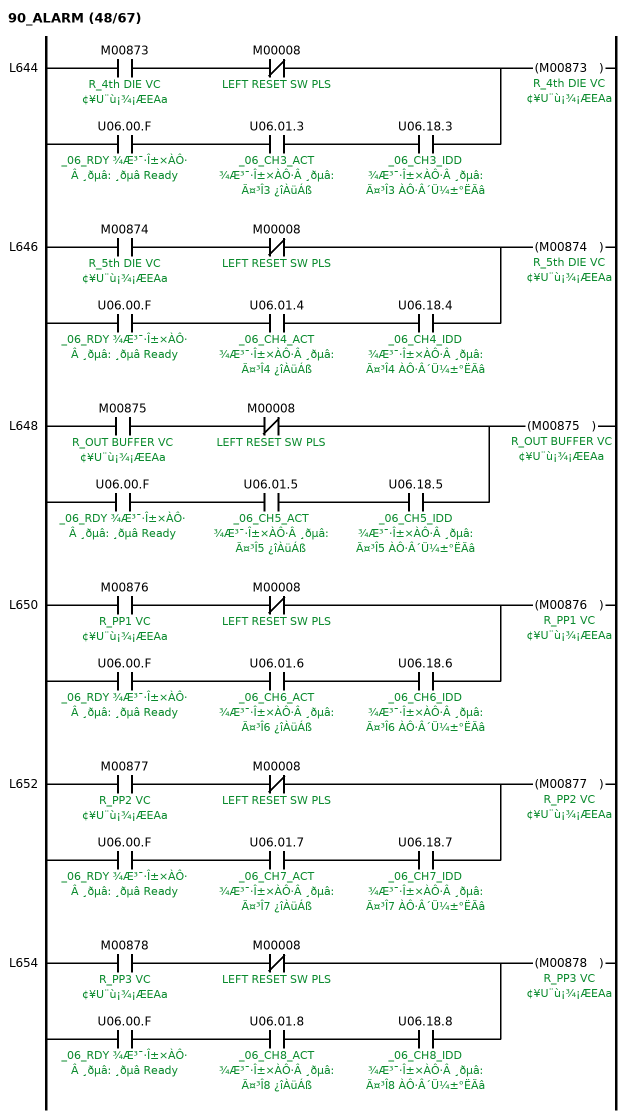
; L644
LOAD      M00873	// R_4th DIE VC ¢¥U¨ù¡¾¡ÆEAa
AND NOT   M00008	// LEFT RESET SW PLS
LOAD      U06.00.F	// _06_RDY ¾Æ³¯·Î±×ÀÔ·Â ¸ðµâ: ¸ðµâ Ready
AND       U06.01.3	// _06_CH3_ACT ¾Æ³¯·Î±×ÀÔ·Â ¸ðµâ: Ã¤³Î3 ¿îÀüÁß
AND       U06.18.3	// _06_CH3_IDD ¾Æ³¯·Î±×ÀÔ·Â ¸ðµâ: Ã¤³Î3 ÀÔ·Â´Ü¼±°ËÃâ
OR LOAD
OUT       M00873	// R_4th DIE VC ¢¥U¨ù¡¾¡ÆEAa
; L646
LOAD      M00874	// R_5th DIE VC ¢¥U¨ù¡¾¡ÆEAa
AND NOT   M00008	// LEFT RESET SW PLS
LOAD      U06.00.F	// _06_RDY ¾Æ³¯·Î±×ÀÔ·Â ¸ðµâ: ¸ðµâ Ready
AND       U06.01.4	// _06_CH4_ACT ¾Æ³¯·Î±×ÀÔ·Â ¸ðµâ: Ã¤³Î4 ¿îÀüÁß
AND       U06.18.4	// _06_CH4_IDD ¾Æ³¯·Î±×ÀÔ·Â ¸ðµâ: Ã¤³Î4 ÀÔ·Â´Ü¼±°ËÃâ
OR LOAD
OUT       M00874	// R_5th DIE VC ¢¥U¨ù¡¾¡ÆEAa
; L648
LOAD      M00875	// R_OUT BUFFER VC ¢¥U¨ù¡¾¡ÆEAa
AND NOT   M00008	// LEFT RESET SW PLS
LOAD      U06.00.F	// _06_RDY ¾Æ³¯·Î±×ÀÔ·Â ¸ðµâ: ¸ðµâ Ready
AND       U06.01.5	// _06_CH5_ACT ¾Æ³¯·Î±×ÀÔ·Â ¸ðµâ: Ã¤³Î5 ¿îÀüÁß
AND       U06.18.5	// _06_CH5_IDD ¾Æ³¯·Î±×ÀÔ·Â ¸ðµâ: Ã¤³Î5 ÀÔ·Â´Ü¼±°ËÃâ
OR LOAD
OUT       M00875	// R_OUT BUFFER VC ¢¥U¨ù¡¾¡ÆEAa
; L650
LOAD      M00876	// R_PP1 VC ¢¥U¨ù¡¾¡ÆEAa
AND NOT   M00008	// LEFT RESET SW PLS
LOAD      U06.00.F	// _06_RDY ¾Æ³¯·Î±×ÀÔ·Â ¸ðµâ: ¸ðµâ Ready
AND       U06.01.6	// _06_CH6_ACT ¾Æ³¯·Î±×ÀÔ·Â ¸ðµâ: Ã¤³Î6 ¿îÀüÁß
AND       U06.18.6	// _06_CH6_IDD ¾Æ³¯·Î±×ÀÔ·Â ¸ðµâ: Ã¤³Î6 ÀÔ·Â´Ü¼±°ËÃâ
OR LOAD
OUT       M00876	// R_PP1 VC ¢¥U¨ù¡¾¡ÆEAa
; L652
LOAD      M00877	// R_PP2 VC ¢¥U¨ù¡¾¡ÆEAa
AND NOT   M00008	// LEFT RESET SW PLS
LOAD      U06.00.F	// _06_RDY ¾Æ³¯·Î±×ÀÔ·Â ¸ðµâ: ¸ðµâ Ready
AND       U06.01.7	// _06_CH7_ACT ¾Æ³¯·Î±×ÀÔ·Â ¸ðµâ: Ã¤³Î7 ¿îÀüÁß
AND       U06.18.7	// _06_CH7_IDD ¾Æ³¯·Î±×ÀÔ·Â ¸ðµâ: Ã¤³Î7 ÀÔ·Â´Ü¼±°ËÃâ
OR LOAD
OUT       M00877	// R_PP2 VC ¢¥U¨ù¡¾¡ÆEAa
; L654
LOAD      M00878	// R_PP3 VC ¢¥U¨ù¡¾¡ÆEAa
AND NOT   M00008	// LEFT RESET SW PLS
LOAD      U06.00.F	// _06_RDY ¾Æ³¯·Î±×ÀÔ·Â ¸ðµâ: ¸ðµâ Ready
AND       U06.01.8	// _06_CH8_ACT ¾Æ³¯·Î±×ÀÔ·Â ¸ðµâ: Ã¤³Î8 ¿îÀüÁß
AND       U06.18.8	// _06_CH8_IDD ¾Æ³¯·Î±×ÀÔ·Â ¸ðµâ: Ã¤³Î8 ÀÔ·Â´Ü¼±°ËÃâ
OR LOAD
OUT       M00878	// R_PP3 VC ¢¥U¨ù¡¾¡ÆEAa

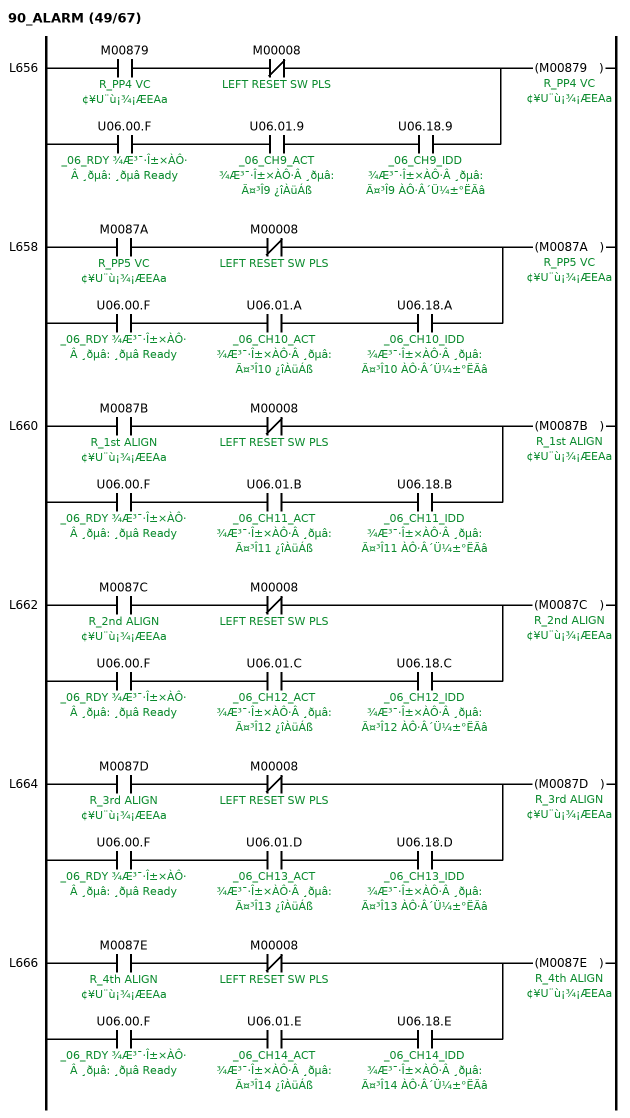
; L656
LOAD      M00879	// R_PP4 VC ¢¥U¨ù¡¾¡ÆEAa
AND NOT   M00008	// LEFT RESET SW PLS
LOAD      U06.00.F	// _06_RDY ¾Æ³¯·Î±×ÀÔ·Â ¸ðµâ: ¸ðµâ Ready
AND       U06.01.9	// _06_CH9_ACT ¾Æ³¯·Î±×ÀÔ·Â ¸ðµâ: Ã¤³Î9 ¿îÀüÁß
AND       U06.18.9	// _06_CH9_IDD ¾Æ³¯·Î±×ÀÔ·Â ¸ðµâ: Ã¤³Î9 ÀÔ·Â´Ü¼±°ËÃâ
OR LOAD
OUT       M00879	// R_PP4 VC ¢¥U¨ù¡¾¡ÆEAa
; L658
LOAD      M0087A	// R_PP5 VC ¢¥U¨ù¡¾¡ÆEAa
AND NOT   M00008	// LEFT RESET SW PLS
LOAD      U06.00.F	// _06_RDY ¾Æ³¯·Î±×ÀÔ·Â ¸ðµâ: ¸ðµâ Ready
AND       U06.01.A	// _06_CH10_ACT ¾Æ³¯·Î±×ÀÔ·Â ¸ðµâ: Ã¤³Î10 ¿îÀüÁß
AND       U06.18.A	// _06_CH10_IDD ¾Æ³¯·Î±×ÀÔ·Â ¸ðµâ: Ã¤³Î10 ÀÔ·Â´Ü¼±°ËÃâ
OR LOAD
OUT       M0087A	// R_PP5 VC ¢¥U¨ù¡¾¡ÆEAa
; L660
LOAD      M0087B	// R_1st ALIGN ¢¥U¨ù¡¾¡ÆEAa
AND NOT   M00008	// LEFT RESET SW PLS
LOAD      U06.00.F	// _06_RDY ¾Æ³¯·Î±×ÀÔ·Â ¸ðµâ: ¸ðµâ Ready
AND       U06.01.B	// _06_CH11_ACT ¾Æ³¯·Î±×ÀÔ·Â ¸ðµâ: Ã¤³Î11 ¿îÀüÁß
AND       U06.18.B	// _06_CH11_IDD ¾Æ³¯·Î±×ÀÔ·Â ¸ðµâ: Ã¤³Î11 ÀÔ·Â´Ü¼±°ËÃâ
OR LOAD
OUT       M0087B	// R_1st ALIGN ¢¥U¨ù¡¾¡ÆEAa
; L662
LOAD      M0087C	// R_2nd ALIGN ¢¥U¨ù¡¾¡ÆEAa
AND NOT   M00008	// LEFT RESET SW PLS
LOAD      U06.00.F	// _06_RDY ¾Æ³¯·Î±×ÀÔ·Â ¸ðµâ: ¸ðµâ Ready
AND       U06.01.C	// _06_CH12_ACT ¾Æ³¯·Î±×ÀÔ·Â ¸ðµâ: Ã¤³Î12 ¿îÀüÁß
AND       U06.18.C	// _06_CH12_IDD ¾Æ³¯·Î±×ÀÔ·Â ¸ðµâ: Ã¤³Î12 ÀÔ·Â´Ü¼±°ËÃâ
OR LOAD
OUT       M0087C	// R_2nd ALIGN ¢¥U¨ù¡¾¡ÆEAa
; L664
LOAD      M0087D	// R_3rd ALIGN ¢¥U¨ù¡¾¡ÆEAa
AND NOT   M00008	// LEFT RESET SW PLS
LOAD      U06.00.F	// _06_RDY ¾Æ³¯·Î±×ÀÔ·Â ¸ðµâ: ¸ðµâ Ready
AND       U06.01.D	// _06_CH13_ACT ¾Æ³¯·Î±×ÀÔ·Â ¸ðµâ: Ã¤³Î13 ¿îÀüÁß
AND       U06.18.D	// _06_CH13_IDD ¾Æ³¯·Î±×ÀÔ·Â ¸ðµâ: Ã¤³Î13 ÀÔ·Â´Ü¼±°ËÃâ
OR LOAD
OUT       M0087D	// R_3rd ALIGN ¢¥U¨ù¡¾¡ÆEAa
; L666
LOAD      M0087E	// R_4th ALIGN ¢¥U¨ù¡¾¡ÆEAa
AND NOT   M00008	// LEFT RESET SW PLS
LOAD      U06.00.F	// _06_RDY ¾Æ³¯·Î±×ÀÔ·Â ¸ðµâ: ¸ðµâ Ready
AND       U06.01.E	// _06_CH14_ACT ¾Æ³¯·Î±×ÀÔ·Â ¸ðµâ: Ã¤³Î14 ¿îÀüÁß
AND       U06.18.E	// _06_CH14_IDD ¾Æ³¯·Î±×ÀÔ·Â ¸ðµâ: Ã¤³Î14 ÀÔ·Â´Ü¼±°ËÃâ
OR LOAD
OUT       M0087E	// R_4th ALIGN ¢¥U¨ù¡¾¡ÆEAa

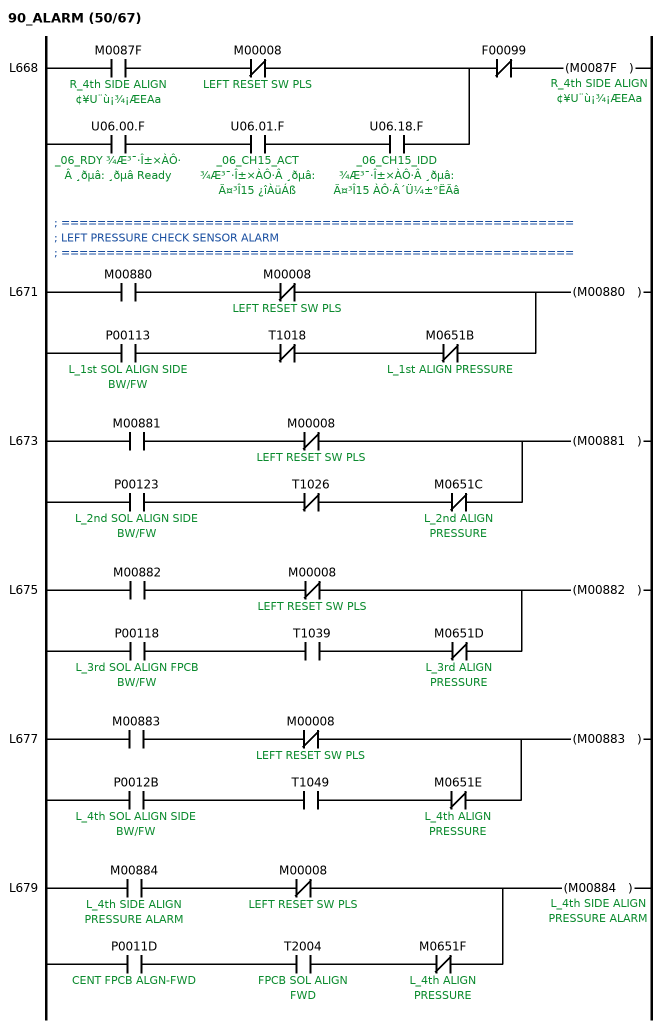
; L668
LOAD      M0087F	// R_4th SIDE ALIGN ¢¥U¨ù¡¾¡ÆEAa
AND NOT   M00008	// LEFT RESET SW PLS
LOAD      U06.00.F	// _06_RDY ¾Æ³¯·Î±×ÀÔ·Â ¸ðµâ: ¸ðµâ Ready
AND       U06.01.F	// _06_CH15_ACT ¾Æ³¯·Î±×ÀÔ·Â ¸ðµâ: Ã¤³Î15 ¿îÀüÁß
AND       U06.18.F	// _06_CH15_IDD ¾Æ³¯·Î±×ÀÔ·Â ¸ðµâ: Ã¤³Î15 ÀÔ·Â´Ü¼±°ËÃâ
OR LOAD
AND NOT   F00099
OUT       M0087F	// R_4th SIDE ALIGN ¢¥U¨ù¡¾¡ÆEAa
// =========================================================
// 
//        LEFT PRESSURE CHECK SENSOR ALARM
// 
// =========================================================
; L671
LOAD      M00880
AND NOT   M00008	// LEFT RESET SW PLS
LOAD      P00113	// L_1st SOL ALIGN SIDE BW/FW
AND NOT   T1018
AND NOT   M0651B	// L_1st ALIGN PRESSURE
OR LOAD
OUT       M00880
; L673
LOAD      M00881
AND NOT   M00008	// LEFT RESET SW PLS
LOAD      P00123	// L_2nd SOL ALIGN SIDE BW/FW
AND NOT   T1026
AND NOT   M0651C	// L_2nd ALIGN PRESSURE
OR LOAD
OUT       M00881
; L675
LOAD      M00882
AND NOT   M00008	// LEFT RESET SW PLS
LOAD      P00118	// L_3rd SOL ALIGN FPCB BW/FW
AND       T1039
AND NOT   M0651D	// L_3rd ALIGN PRESSURE
OR LOAD
OUT       M00882
; L677
LOAD      M00883
AND NOT   M00008	// LEFT RESET SW PLS
LOAD      P0012B	// L_4th SOL ALIGN SIDE BW/FW
AND       T1049
AND NOT   M0651E	// L_4th ALIGN PRESSURE
OR LOAD
OUT       M00883
; L679
LOAD      M00884	// L_4th SIDE ALIGN PRESSURE ALARM
AND NOT   M00008	// LEFT RESET SW PLS
LOAD      P0011D	// CENT FPCB ALGN-FWD
AND       T2004	// FPCB SOL ALIGN         FWD
AND NOT   M0651F	// L_4th ALIGN PRESSURE
OR LOAD
OUT       M00884	// L_4th SIDE ALIGN PRESSURE ALARM

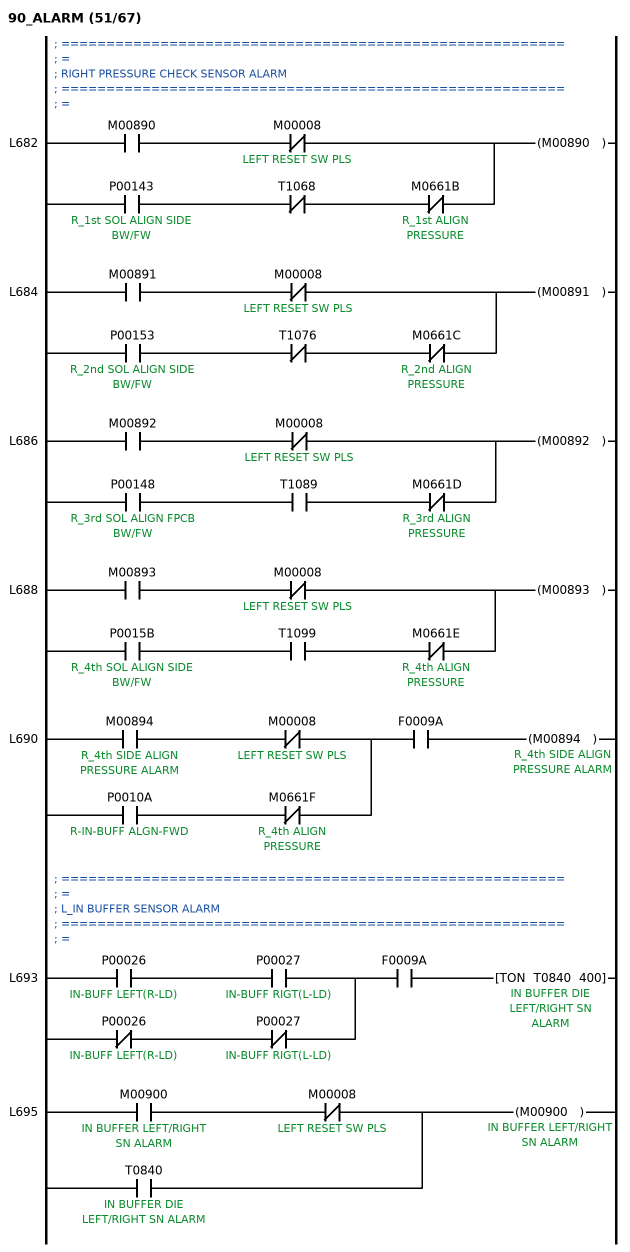
// =========================================================
// 
//        RIGHT PRESSURE CHECK SENSOR ALARM
// 
// =========================================================
; L682
LOAD      M00890
AND NOT   M00008	// LEFT RESET SW PLS
LOAD      P00143	// R_1st SOL ALIGN SIDE BW/FW
AND NOT   T1068
AND NOT   M0661B	// R_1st ALIGN PRESSURE
OR LOAD
OUT       M00890
; L684
LOAD      M00891
AND NOT   M00008	// LEFT RESET SW PLS
LOAD      P00153	// R_2nd SOL ALIGN SIDE BW/FW
AND NOT   T1076
AND NOT   M0661C	// R_2nd ALIGN PRESSURE
OR LOAD
OUT       M00891
; L686
LOAD      M00892
AND NOT   M00008	// LEFT RESET SW PLS
LOAD      P00148	// R_3rd SOL ALIGN FPCB BW/FW
AND       T1089
AND NOT   M0661D	// R_3rd ALIGN PRESSURE
OR LOAD
OUT       M00892
; L688
LOAD      M00893
AND NOT   M00008	// LEFT RESET SW PLS
LOAD      P0015B	// R_4th SOL ALIGN SIDE BW/FW
AND       T1099
AND NOT   M0661E	// R_4th ALIGN PRESSURE
OR LOAD
OUT       M00893
; L690
LOAD      M00894	// R_4th SIDE ALIGN PRESSURE ALARM
AND NOT   M00008	// LEFT RESET SW PLS
LOAD      P0010A	// R-IN-BUFF ALGN-FWD
AND NOT   M0661F	// R_4th ALIGN PRESSURE
OR LOAD
AND       F0009A
OUT       M00894	// R_4th SIDE ALIGN PRESSURE ALARM
// =========================================================
// 
//        L_IN BUFFER SENSOR ALARM
// 
// =========================================================
; L693
LOAD      P00026	// IN-BUFF LEFT(R-LD)
AND       P00027	// IN-BUFF RIGT(L-LD)
LOAD NOT  P00026	// IN-BUFF LEFT(R-LD)
AND NOT   P00027	// IN-BUFF RIGT(L-LD)
OR LOAD
AND       F0009A
TON       T0840 400	// IN BUFFER DIE LEFT/RIGHT SN ALARM
; L695
LOAD      M00900	// IN BUFFER LEFT/RIGHT SN ALARM
AND NOT   M00008	// LEFT RESET SW PLS
OR        T0840	// IN BUFFER DIE LEFT/RIGHT SN ALARM
OUT       M00900	// IN BUFFER LEFT/RIGHT SN ALARM

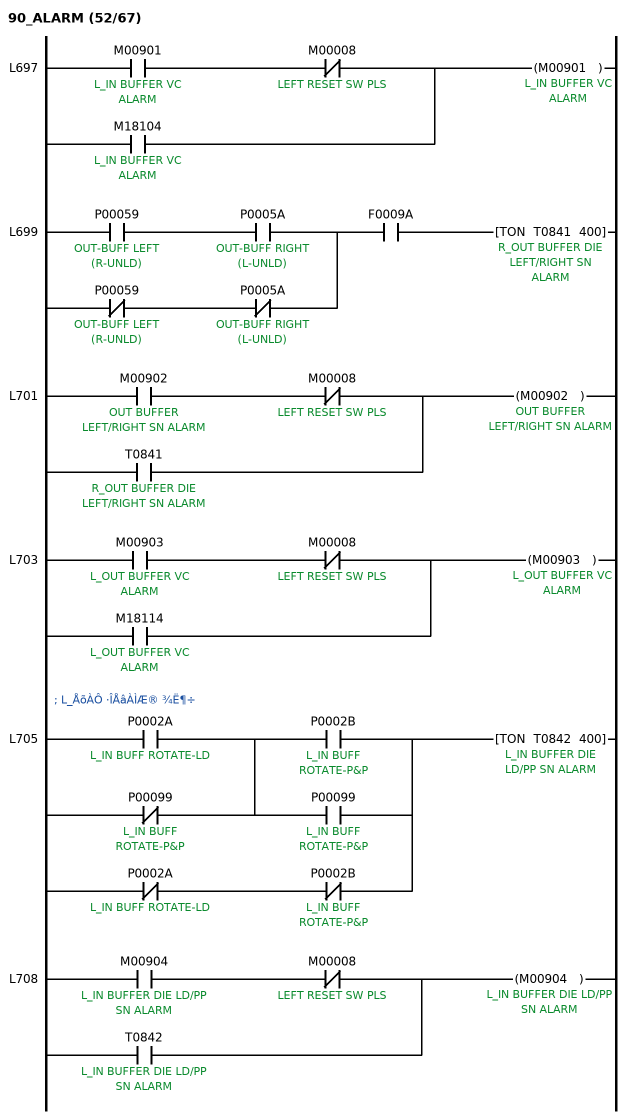
; L697
LOAD      M00901	// L_IN BUFFER VC ALARM
AND NOT   M00008	// LEFT RESET SW PLS
OR        M18104	// L_IN BUFFER VC ALARM
OUT       M00901	// L_IN BUFFER VC ALARM
; L699
LOAD      P00059	// OUT-BUFF LEFT (R-UNLD)
AND       P0005A	// OUT-BUFF RIGHT (L-UNLD)
LOAD NOT  P00059	// OUT-BUFF LEFT (R-UNLD)
AND NOT   P0005A	// OUT-BUFF RIGHT (L-UNLD)
OR LOAD
AND       F0009A
TON       T0841 400	// R_OUT BUFFER DIE LEFT/RIGHT SN ALARM
; L701
LOAD      M00902	// OUT BUFFER LEFT/RIGHT SN ALARM
AND NOT   M00008	// LEFT RESET SW PLS
OR        T0841	// R_OUT BUFFER DIE LEFT/RIGHT SN ALARM
OUT       M00902	// OUT BUFFER LEFT/RIGHT SN ALARM
; L703
LOAD      M00903	// L_OUT BUFFER VC ALARM
AND NOT   M00008	// LEFT RESET SW PLS
OR        M18114	// L_OUT BUFFER VC ALARM
OUT       M00903	// L_OUT BUFFER VC ALARM
; L705
LOAD      P0002A	// L_IN BUFF ROTATE-LD
OR NOT    P00099	// L_IN BUFF ROTATE-P&P
LOAD      P0002B	// L_IN BUFF ROTATE-P&P
OR        P00099	// L_IN BUFF ROTATE-P&P
AND LOAD
LOAD NOT  P0002A	// L_IN BUFF ROTATE-LD
AND NOT   P0002B	// L_IN BUFF ROTATE-P&P
OR LOAD
TON       T0842 400	// L_IN BUFFER DIE LD/PP SN ALARM
// output comment: L_ÅõÀÔ ·ÎÅâÀÌÆ® ¾Ë¶÷
; L708
LOAD      M00904	// L_IN BUFFER DIE LD/PP SN ALARM
AND NOT   M00008	// LEFT RESET SW PLS
OR        T0842	// L_IN BUFFER DIE LD/PP SN ALARM
OUT       M00904	// L_IN BUFFER DIE LD/PP SN ALARM

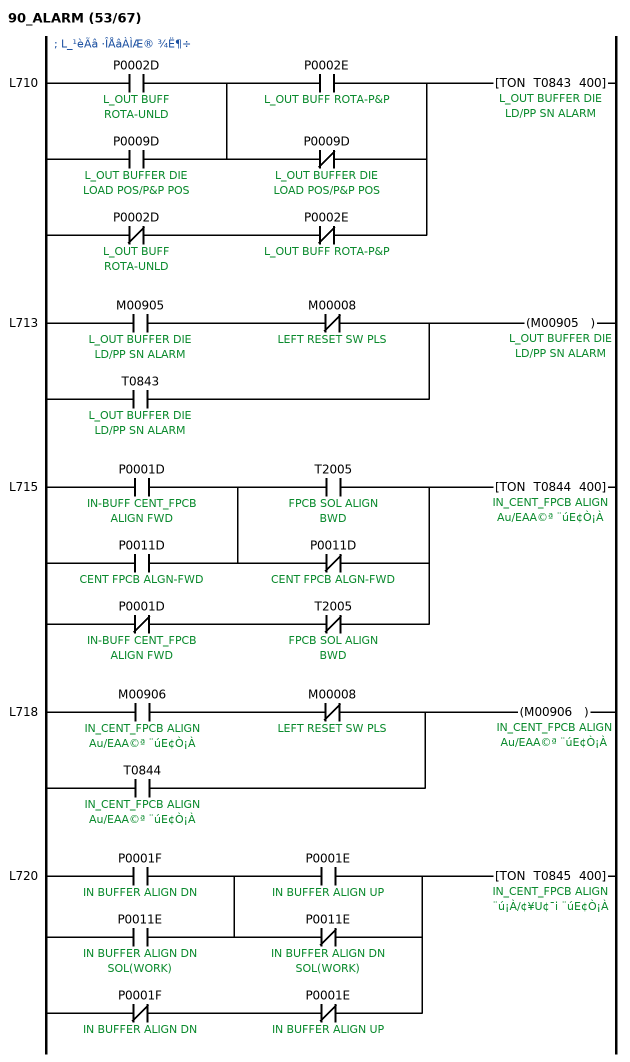
; L710
LOAD      P0002D	// L_OUT BUFF ROTA-UNLD
OR        P0009D	// L_OUT BUFFER DIE LOAD POS/P&P POS
LOAD      P0002E	// L_OUT BUFF ROTA-P&P
OR NOT    P0009D	// L_OUT BUFFER DIE LOAD POS/P&P POS
AND LOAD
LOAD NOT  P0002D	// L_OUT BUFF ROTA-UNLD
AND NOT   P0002E	// L_OUT BUFF ROTA-P&P
OR LOAD
TON       T0843 400	// L_OUT BUFFER DIE LD/PP SN ALARM
// output comment: L_¹èÃâ ·ÎÅâÀÌÆ® ¾Ë¶÷
; L713
LOAD      M00905	// L_OUT BUFFER DIE LD/PP SN ALARM
AND NOT   M00008	// LEFT RESET SW PLS
OR        T0843	// L_OUT BUFFER DIE LD/PP SN ALARM
OUT       M00905	// L_OUT BUFFER DIE LD/PP SN ALARM
; L715
LOAD      P0001D	// IN-BUFF CENT_FPCB ALIGN FWD
OR        P0011D	// CENT FPCB ALGN-FWD
LOAD      T2005	// FPCB SOL ALIGN         BWD
OR NOT    P0011D	// CENT FPCB ALGN-FWD
AND LOAD
LOAD NOT  P0001D	// IN-BUFF CENT_FPCB ALIGN FWD
AND NOT   T2005	// FPCB SOL ALIGN         BWD
OR LOAD
TON       T0844 400	// IN_CENT_FPCB ALIGN Au/EAA©ª ¨úE¢Ò¡À
; L718
LOAD      M00906	// IN_CENT_FPCB ALIGN Au/EAA©ª ¨úE¢Ò¡À
AND NOT   M00008	// LEFT RESET SW PLS
OR        T0844	// IN_CENT_FPCB ALIGN Au/EAA©ª ¨úE¢Ò¡À
OUT       M00906	// IN_CENT_FPCB ALIGN Au/EAA©ª ¨úE¢Ò¡À
; L720
LOAD      P0001F	// IN BUFFER ALIGN DN
OR        P0011E	// IN BUFFER ALIGN DN SOL(WORK)
LOAD      P0001E	// IN BUFFER ALIGN UP
OR NOT    P0011E	// IN BUFFER ALIGN DN SOL(WORK)
AND LOAD
LOAD NOT  P0001F	// IN BUFFER ALIGN DN
AND NOT   P0001E	// IN BUFFER ALIGN UP
OR LOAD
TON       T0845 400	// IN_CENT_FPCB ALIGN ¨ú¡À/¢¥U¢¯i ¨úE¢Ò¡À

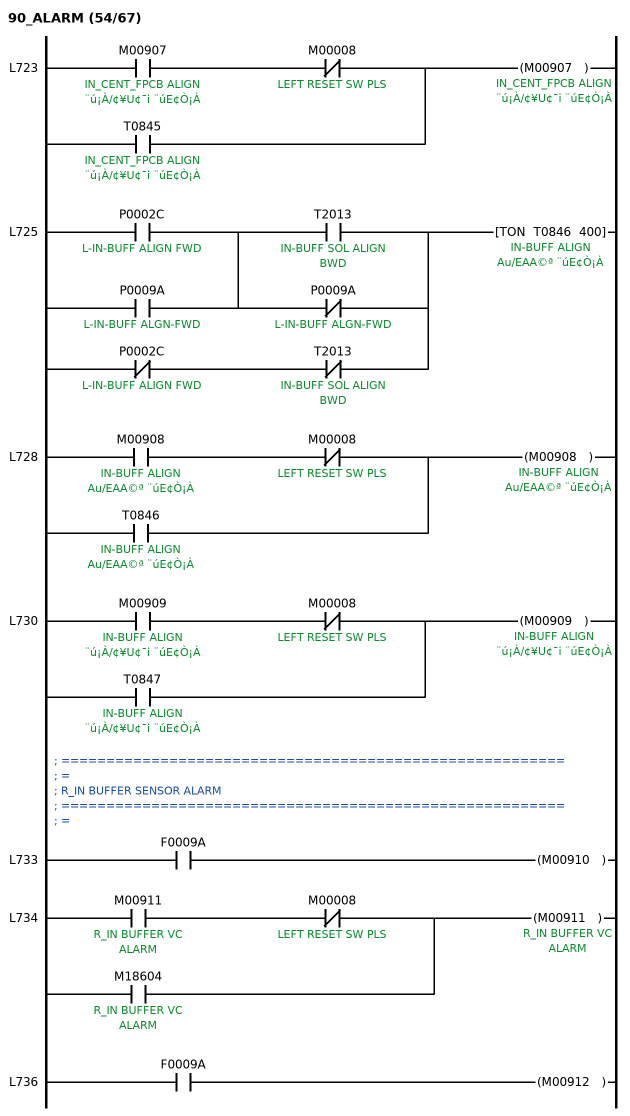
; L723
LOAD      M00907	// IN_CENT_FPCB ALIGN ¨ú¡À/¢¥U¢¯i ¨úE¢Ò¡À
AND NOT   M00008	// LEFT RESET SW PLS
OR        T0845	// IN_CENT_FPCB ALIGN ¨ú¡À/¢¥U¢¯i ¨úE¢Ò¡À
OUT       M00907	// IN_CENT_FPCB ALIGN ¨ú¡À/¢¥U¢¯i ¨úE¢Ò¡À
; L725
LOAD      P0002C	// L-IN-BUFF ALIGN FWD
OR        P0009A	// L-IN-BUFF ALGN-FWD
LOAD      T2013	// IN-BUFF SOL ALIGN BWD
OR NOT    P0009A	// L-IN-BUFF ALGN-FWD
AND LOAD
LOAD NOT  P0002C	// L-IN-BUFF ALIGN FWD
AND NOT   T2013	// IN-BUFF SOL ALIGN BWD
OR LOAD
TON       T0846 400	// IN-BUFF ALIGN Au/EAA©ª ¨úE¢Ò¡À
; L728
LOAD      M00908	// IN-BUFF ALIGN Au/EAA©ª ¨úE¢Ò¡À
AND NOT   M00008	// LEFT RESET SW PLS
OR        T0846	// IN-BUFF ALIGN Au/EAA©ª ¨úE¢Ò¡À
OUT       M00908	// IN-BUFF ALIGN Au/EAA©ª ¨úE¢Ò¡À
; L730
LOAD      M00909	// IN-BUFF ALIGN ¨ú¡À/¢¥U¢¯i ¨úE¢Ò¡À
AND NOT   M00008	// LEFT RESET SW PLS
OR        T0847	// IN-BUFF ALIGN ¨ú¡À/¢¥U¢¯i ¨úE¢Ò¡À
OUT       M00909	// IN-BUFF ALIGN ¨ú¡À/¢¥U¢¯i ¨úE¢Ò¡À
// =========================================================
// 
//        R_IN BUFFER SENSOR ALARM
// 
// =========================================================
; L733
LOAD      F0009A
OUT       M00910
; L734
LOAD      M00911	// R_IN BUFFER VC ALARM
AND NOT   M00008	// LEFT RESET SW PLS
OR        M18604	// R_IN BUFFER VC ALARM
OUT       M00911	// R_IN BUFFER VC ALARM
; L736
LOAD      F0009A
OUT       M00912

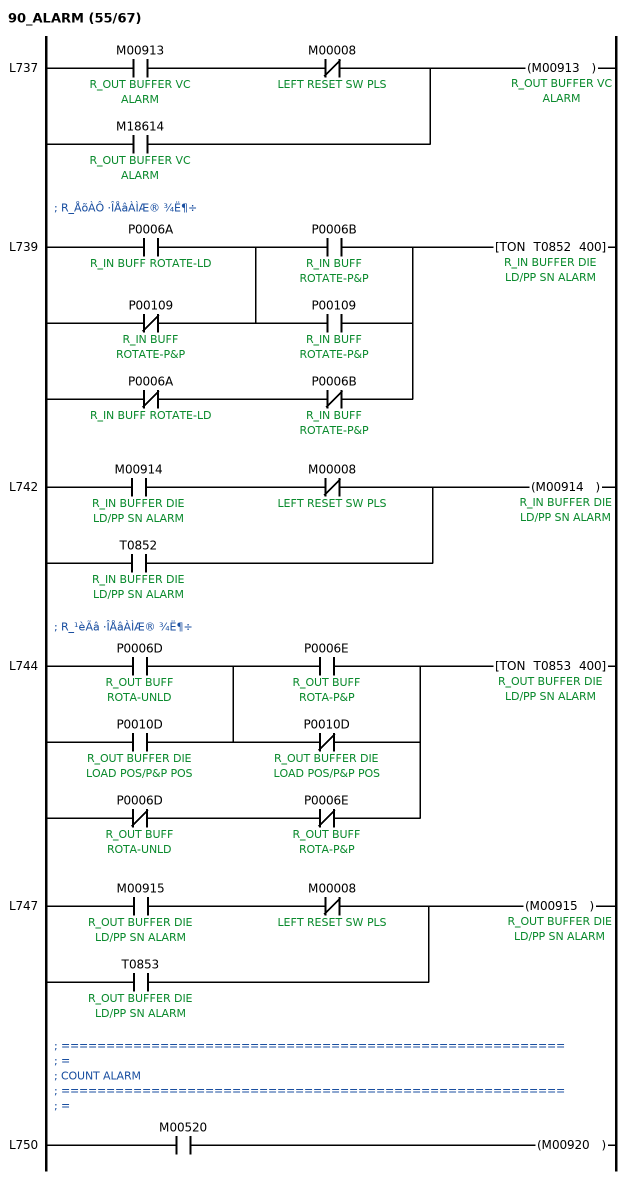
; L737
LOAD      M00913	// R_OUT BUFFER VC ALARM
AND NOT   M00008	// LEFT RESET SW PLS
OR        M18614	// R_OUT BUFFER VC ALARM
OUT       M00913	// R_OUT BUFFER VC ALARM
; L739
LOAD      P0006A	// R_IN BUFF ROTATE-LD
OR NOT    P00109	// R_IN BUFF ROTATE-P&P
LOAD      P0006B	// R_IN BUFF ROTATE-P&P
OR        P00109	// R_IN BUFF ROTATE-P&P
AND LOAD
LOAD NOT  P0006A	// R_IN BUFF ROTATE-LD
AND NOT   P0006B	// R_IN BUFF ROTATE-P&P
OR LOAD
TON       T0852 400	// R_IN BUFFER DIE LD/PP SN ALARM
// output comment: R_ÅõÀÔ ·ÎÅâÀÌÆ® ¾Ë¶÷
; L742
LOAD      M00914	// R_IN BUFFER DIE LD/PP SN ALARM
AND NOT   M00008	// LEFT RESET SW PLS
OR        T0852	// R_IN BUFFER DIE LD/PP SN ALARM
OUT       M00914	// R_IN BUFFER DIE LD/PP SN ALARM
; L744
LOAD      P0006D	// R_OUT BUFF ROTA-UNLD
OR        P0010D	// R_OUT BUFFER DIE LOAD POS/P&P POS
LOAD      P0006E	// R_OUT BUFF ROTA-P&P
OR NOT    P0010D	// R_OUT BUFFER DIE LOAD POS/P&P POS
AND LOAD
LOAD NOT  P0006D	// R_OUT BUFF ROTA-UNLD
AND NOT   P0006E	// R_OUT BUFF ROTA-P&P
OR LOAD
TON       T0853 400	// R_OUT BUFFER DIE LD/PP SN ALARM
// output comment: R_¹èÃâ ·ÎÅâÀÌÆ® ¾Ë¶÷
; L747
LOAD      M00915	// R_OUT BUFFER DIE LD/PP SN ALARM
AND NOT   M00008	// LEFT RESET SW PLS
OR        T0853	// R_OUT BUFFER DIE LD/PP SN ALARM
OUT       M00915	// R_OUT BUFFER DIE LD/PP SN ALARM
// =========================================================
// 
//       COUNT ALARM
// 
// =========================================================
; L750
LOAD      M00520
OUT       M00920

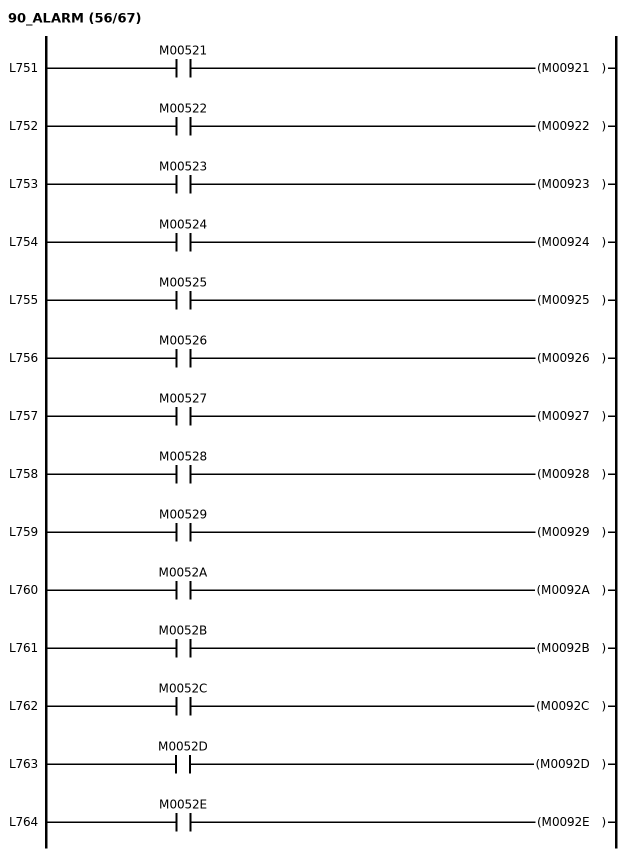
; L751
LOAD      M00521
OUT       M00921
; L752
LOAD      M00522
OUT       M00922
; L753
LOAD      M00523
OUT       M00923
; L754
LOAD      M00524
OUT       M00924
; L755
LOAD      M00525
OUT       M00925
; L756
LOAD      M00526
OUT       M00926
; L757
LOAD      M00527
OUT       M00927
; L758
LOAD      M00528
OUT       M00928
; L759
LOAD      M00529
OUT       M00929
; L760
LOAD      M0052A
OUT       M0092A
; L761
LOAD      M0052B
OUT       M0092B
; L762
LOAD      M0052C
OUT       M0092C
; L763
LOAD      M0052D
OUT       M0092D
; L764
LOAD      M0052E
OUT       M0092E

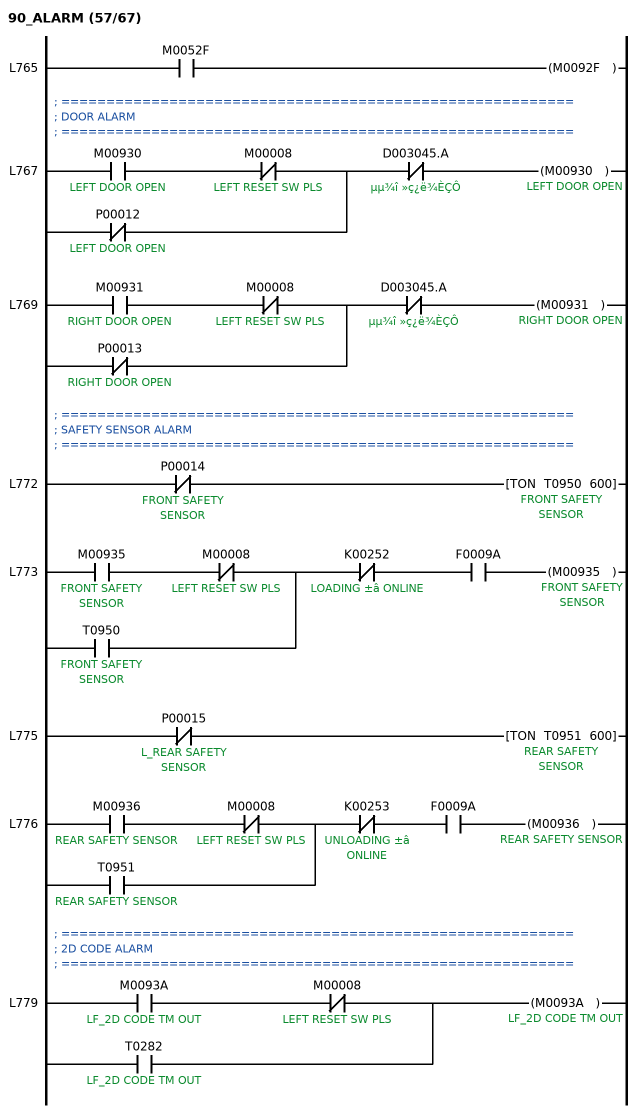
; L765
LOAD      M0052F
OUT       M0092F
// =========================================================
// 
//       DOOR ALARM
// 
// =========================================================
; L767
LOAD      M00930	// LEFT DOOR OPEN
AND NOT   M00008	// LEFT RESET SW PLS
OR NOT    P00012	// LEFT DOOR OPEN
AND NOT   D003045.A	// µµ¾î »ç¿ë¾ÈÇÔ
OUT       M00930	// LEFT DOOR OPEN
; L769
LOAD      M00931	// RIGHT DOOR OPEN
AND NOT   M00008	// LEFT RESET SW PLS
OR NOT    P00013	// RIGHT DOOR OPEN
AND NOT   D003045.A	// µµ¾î »ç¿ë¾ÈÇÔ
OUT       M00931	// RIGHT DOOR OPEN
// =========================================================
// 
//       SAFETY SENSOR ALARM
// 
// =========================================================
; L772
LOAD NOT  P00014	// FRONT SAFETY SENSOR
TON       T0950 600	// FRONT SAFETY SENSOR
; L773
LOAD      M00935	// FRONT SAFETY SENSOR
AND NOT   M00008	// LEFT RESET SW PLS
OR        T0950	// FRONT SAFETY SENSOR
AND NOT   K00252	// LOADING ±â ONLINE
AND       F0009A
OUT       M00935	// FRONT SAFETY SENSOR
; L775
LOAD NOT  P00015	// L_REAR SAFETY SENSOR
TON       T0951 600	// REAR SAFETY SENSOR
; L776
LOAD      M00936	// REAR SAFETY SENSOR
AND NOT   M00008	// LEFT RESET SW PLS
OR        T0951	// REAR SAFETY SENSOR
AND NOT   K00253	// UNLOADING ±â ONLINE
AND       F0009A
OUT       M00936	// REAR SAFETY SENSOR
// =========================================================
// 
//       2D CODE ALARM
// 
// =========================================================
; L779
LOAD      M0093A	// LF_2D CODE TM OUT
AND NOT   M00008	// LEFT RESET SW PLS
OR        T0282	// LF_2D CODE TM OUT
OUT       M0093A	// LF_2D CODE TM OUT

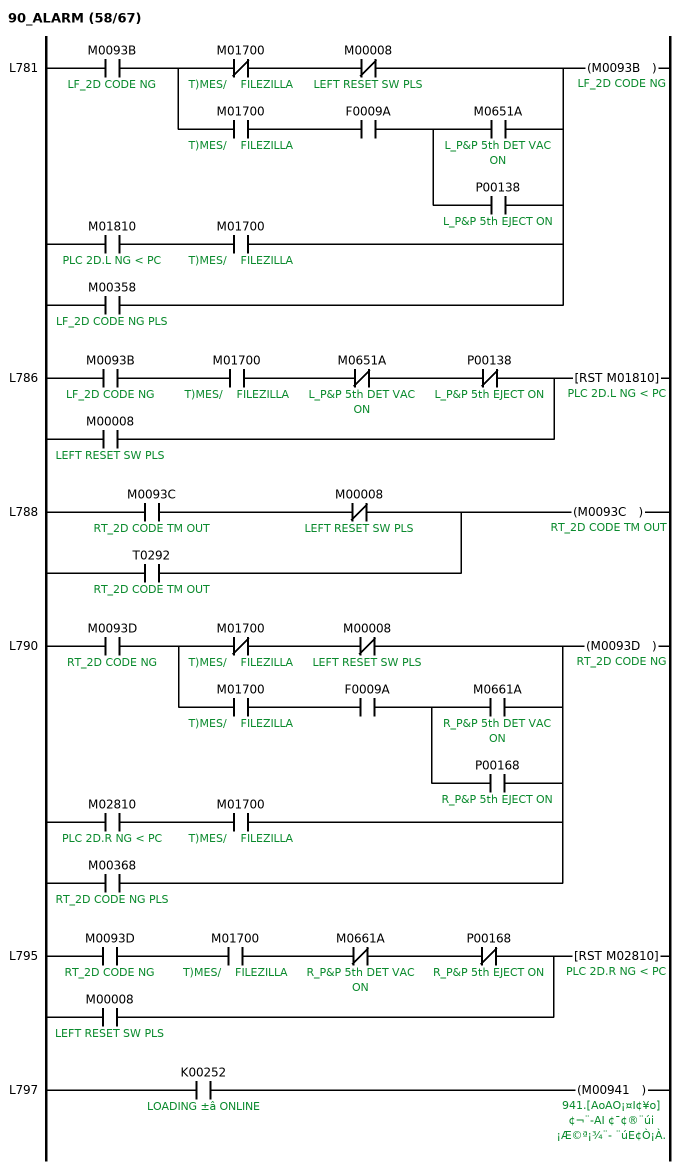
; L781
LOAD      M0093B	// LF_2D CODE NG
LOAD NOT  M01700	// T)MES/    FILEZILLA
AND NOT   M00008	// LEFT RESET SW PLS
LOAD      M01700	// T)MES/    FILEZILLA
AND       F0009A
LOAD      M0651A	// L_P&P 5th DET VAC ON
OR        P00138	// L_P&P 5th EJECT ON
AND LOAD
OR LOAD
AND LOAD
LOAD      M01810	// PLC 2D.L NG < PC
AND       M01700	// T)MES/    FILEZILLA
OR LOAD
OR        M00358	// LF_2D CODE NG PLS
OUT       M0093B	// LF_2D CODE NG
; L786
LOAD      M0093B	// LF_2D CODE NG
AND       M01700	// T)MES/    FILEZILLA
AND NOT   M0651A	// L_P&P 5th DET VAC ON
AND NOT   P00138	// L_P&P 5th EJECT ON
OR        M00008	// LEFT RESET SW PLS
RST       M01810	// PLC 2D.L NG < PC
; L788
LOAD      M0093C	// RT_2D CODE TM OUT
AND NOT   M00008	// LEFT RESET SW PLS
OR        T0292	// RT_2D CODE TM OUT
OUT       M0093C	// RT_2D CODE TM OUT
; L790
LOAD      M0093D	// RT_2D CODE NG
LOAD NOT  M01700	// T)MES/    FILEZILLA
AND NOT   M00008	// LEFT RESET SW PLS
LOAD      M01700	// T)MES/    FILEZILLA
AND       F0009A
LOAD      M0661A	// R_P&P 5th DET VAC ON
OR        P00168	// R_P&P 5th EJECT ON
AND LOAD
OR LOAD
AND LOAD
LOAD      M02810	// PLC 2D.R NG < PC
AND       M01700	// T)MES/    FILEZILLA
OR LOAD
OR        M00368	// RT_2D CODE NG PLS
OUT       M0093D	// RT_2D CODE NG
; L795
LOAD      M0093D	// RT_2D CODE NG
AND       M01700	// T)MES/    FILEZILLA
AND NOT   M0661A	// R_P&P 5th DET VAC ON
AND NOT   P00168	// R_P&P 5th EJECT ON
OR        M00008	// LEFT RESET SW PLS
RST       M02810	// PLC 2D.R NG < PC
; L797
LOAD      K00252	// LOADING ±â ONLINE
OUT       M00941	// 941.[AoAO¡¤I¢¥o] ¢¬¨­AI ¢¯¢®¨úi ¡Æ©ª¡¾¨­ ¨úE¢Ò¡À.

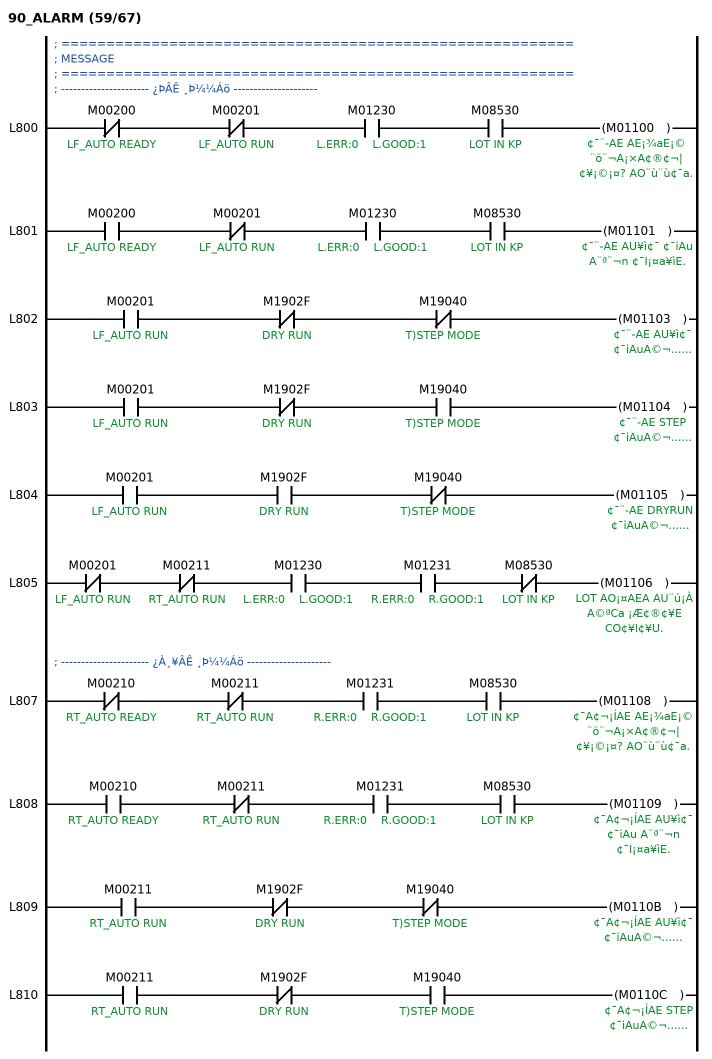
// =========================================================
// 
//       MESSAGE
// 
// =========================================================
// ---------------------- ¿ÞÂÊ ¸Þ¼¼Áö ---------------------
; L800
LOAD NOT  M00200	// LF_AUTO READY
AND NOT   M00201	// LF_AUTO RUN
AND       M01230	// L.ERR:0    L.GOOD:1
AND       M08530	// LOT IN KP
OUT       M01100	// ¢¯¨­AE AE¡¾aE¡© ¨ö¨¬A¡×A¢®¢¬| ¢¥¡©¡¤? AO¨ù¨ù¢¯a.
; L801
LOAD      M00200	// LF_AUTO READY
AND NOT   M00201	// LF_AUTO RUN
AND       M01230	// L.ERR:0    L.GOOD:1
AND       M08530	// LOT IN KP
OUT       M01101	// ¢¯¨­AE AU¥ì¢¯ ¢¯iAu A¨ª¨¬n ¢¯I¡¤a¥ìE.
; L802
LOAD      M00201	// LF_AUTO RUN
AND NOT   M1902F	// DRY RUN
AND NOT   M19040	// T)STEP MODE
OUT       M01103	// ¢¯¨­AE AU¥ì¢¯ ¢¯iAuA©¬......
; L803
LOAD      M00201	// LF_AUTO RUN
AND NOT   M1902F	// DRY RUN
AND       M19040	// T)STEP MODE
OUT       M01104	// ¢¯¨­AE STEP ¢¯iAuA©¬......
; L804
LOAD      M00201	// LF_AUTO RUN
AND       M1902F	// DRY RUN
AND NOT   M19040	// T)STEP MODE
OUT       M01105	// ¢¯¨­AE DRYRUN ¢¯iAuA©¬......
; L805
LOAD NOT  M00201	// LF_AUTO RUN
AND NOT   M00211	// RT_AUTO RUN
AND       M01230	// L.ERR:0    L.GOOD:1
AND       M01231	// R.ERR:0    R.GOOD:1
AND NOT   M08530	// LOT IN KP
OUT       M01106	// LOT AO¡¤AEA AU¨ú¡À A©ªCa ¡Æ¢®¢¥E CO¢¥I¢¥U.
// ---------------------- ¿À¸¥ÂÊ ¸Þ¼¼Áö ---------------------
; L807
LOAD NOT  M00210	// RT_AUTO READY
AND NOT   M00211	// RT_AUTO RUN
AND       M01231	// R.ERR:0    R.GOOD:1
AND       M08530	// LOT IN KP
OUT       M01108	// ¢¯A¢¬¡ÍAE AE¡¾aE¡© ¨ö¨¬A¡×A¢®¢¬| ¢¥¡©¡¤? AO¨ù¨ù¢¯a.
; L808
LOAD      M00210	// RT_AUTO READY
AND NOT   M00211	// RT_AUTO RUN
AND       M01231	// R.ERR:0    R.GOOD:1
AND       M08530	// LOT IN KP
OUT       M01109	// ¢¯A¢¬¡ÍAE AU¥ì¢¯ ¢¯iAu A¨ª¨¬n ¢¯I¡¤a¥ìE.
; L809
LOAD      M00211	// RT_AUTO RUN
AND NOT   M1902F	// DRY RUN
AND NOT   M19040	// T)STEP MODE
OUT       M0110B	// ¢¯A¢¬¡ÍAE AU¥ì¢¯ ¢¯iAuA©¬......
; L810
LOAD      M00211	// RT_AUTO RUN
AND NOT   M1902F	// DRY RUN
AND       M19040	// T)STEP MODE
OUT       M0110C	// ¢¯A¢¬¡ÍAE STEP ¢¯iAuA©¬......

